_mode_manager();

CASE process_get_mode(prc) OF
	MODE_ABSENT:
		IF axis_get_mode(axis) = MODE_TEST
		THEN
			safety_integrated_series_close(csp_transfer_main_safety_drives_SD41100.chA_smes_sis);
		END_IF
		RETURN;
	MODE_INACTIVE:
		RETURN;
	MODE_TEST:
		_handle_process_test();
END_CASE

(********************************* BODY *********************************)
axis.actual_torque := (axis.actual_current * Torque_force_constant)/1000;

(* Sets torque Limit *)
IF torque_limit <> torque_limit_old
THEN
	IF soe_drive_channel_write_parameter(
		channel:= csp_transfer_accumulator_lift.axis.soe_drive_channel, 
		idn:= S_0_IDN + 92, 
		data_element:= soe_drive_element_value, 
		data_source:= ADR(torque_limit), 
		data_lenght:= SIZEOF(torque_limit),
		CONVERSION_this:= csp_transfer_accumulator_lift.axis.soe_drive^) = SOE_DRIVE_RETURN_VALUE_DONE
	THEN
		torque_limit_old := torque_limit;
	END_IF
END_IF

(* Connection Done Test *)
IF connection_done
THEN 
	motorization_conditioner_start_done(connection_done_motcond);
END_IF

(* CLEARS CONNECTION AND PHASE ERRORS *)
IF 	machine_is_stopped(csp.mch)
	OR machine_is_stop_emergency_active(csp.mch)
	OR machine_is_ready(csp.mch)
	OR csp_main_services_pushbuttons.i_reset_button
THEN
	connection_error := FALSE;
	phase_error := FALSE;
END_IF

(* RESETS AXES IF PHASE DONE AND CONNECTION DONE AND DISABLED *)
IF 	phase_done
	AND connection_done
	AND axis_is_disabled(axis)
THEN
	phase_done := FALSE;
	connection_done := FALSE;
END_IF


(* CAM CHANGE/CHECK LOGIC *)
IF 	phase_edge(csp_transfer_crosspusher_virtualMaster.cam_change_check_ph) (* CROSSPUSHER VIRTUAL AT CHECK PHASE DEG *)
	AND connection_status = CSP_TRANSFER_CROSSPUSHER_STATUS_CONNECTION_CHECK_CHANGE_CAM
THEN	
	IF run_test 
	OR
	(
	csp_transfer_upstacker.stack_made (* UPSTACKER MADE CORRECT AMOUNT OF STACK *)
	AND csp_transfer_crosspusher_horizontal.at_upstack (* VERIFIES THE HORIZONTAL IS AT THE UPSTACKER BEFORE RUNNING *)
	AND NOT csp_transfer_upstacker.stack_at_loader (* MAKES SURE A STACK IS NOT ALREADY AT THE LOADER *)
	)
	THEN 
		run := TRUE;
	ELSE
		dwell := TRUE;
	END_IF
END_IF

(* DWELL CAM BECAUSE LOADER NOT CLEAR - IMMEDIATELY *)
IF active_cam = TRANSFER_ACCUMULATOR_LIFT_RUN
	AND csp_transfer_crosspusher.loader_status = csp_transfer_crosspusher_loader_clear_status.NOT_CLEAR 
THEN
	connection_status_next := CSP_TRANSFER_CROSSPUSHER_STATUS_CONNECTION_IMMEDIATE_CHANGE;
	connection_status := CSP_TRANSFER_CROSSPUSHER_STATUS_CONNECTION_IMMEDIATE_CHANGE;
END_IF

(* ERROR HANDLING FOR CAM ERROR *)
IF active_cam = 0
THEN 
	active_cam := DWELL_CAM;
END_IF

(* TELLS THE FOLLOWER WHAT THE PROFILE SHOULD BE ON A CLEARED LOAD *)
IF csp_transfer_upstacker.stack_removed_from_upstack
THEN
	active_cam := DWELL_CAM;
END_IF

(* MAIN ACTIONS IN POU *)
phase();
connection();
_set_runtime_properties();

(************************************************************************)

_handle_messages();

_write_output();

ACTION _handle_messages:
;
END_ACTION

ACTION _handle_process_test:
;
END_ACTION

ACTION _mode_manager:
IF process_mode_req_is_pending(prc)
THEN
    process_apply_mode_req_first_step(prc);
    CASE process_get_mode(prc) OF
        MODE_TO_ABSENT:
			;
        MODE_TO_INACTIVE:
			;
        MODE_TO_TEST:
			;
        MODE_TO_OPERATIONAL:
			;
    END_CASE
    process_apply_mode_req_second_step(prc);
END_IF
END_ACTION

ACTION _object_manager:
IF objects_initialization()
THEN
	sub_process_init(
		object_name					:= 'csp_transfer_accumulator_lift.prc', 
		process						:= csp_transfer_accumulator.prc, 
		CONVERSION_this				:= prc);
		
	prc_path 						:= process_get_path(prc);
	
	axis_init(
		object_name					:= CONCAT(prc_path, '_axis'), 
		axis_type					:= AXIS_TYPE_SERVO, 
		encoder_scaling_factor		:= G_SERVO_ENCODER_SCALING_FACTOR_DEGPINC,
		modulo						:= G_MODULO_360_DEG, 
		process						:= prc, 
		CONVERSION_this				:= axis);
		
	axis_init_absolute_encoder_preset(	
		position					:=	0,
		CONVERSION_this				:=	axis);
	
	axis_set_max_dynamic(
		reference_velocity			:=	MOTOR_MAX_VELOCITY_DEGPS,
		velocity					:=	MOTOR_MAX_VELOCITY_DEGPS,
		acceleration				:=	MOTOR_MAX_ACCELLERATION_DEGPS2,
		deceleration				:=	MOTOR_MAX_DECELLERATION_DEGPS2,
		jerk						:=	MOTOR_MAX_JERK_DEGPS3,
		following_error				:=	MOTOR_MAX_FOLLOWING_ERROR_DEG,
		CONVERSION_this				:=	axis);
	
	axis_add_soe_drive(
		channel						:=	SOE_DRIVE_CHANNEL_A,
		soe_drive					:=	csp_transfer_main_drives.SD41100_drv,
		CONVERSION_this				:=	axis);
		
	process_message_init(
		object_name					:=	CONCAT(prc_path, '_phase_faulted_aem'), 
		behaviour					:=	MESSAGE_BEHAVIOUR_EVENT,
		reset_timeout				:=	0,
		disableable					:=	TRUE,
		individual_reset			:=	FALSE,
		machine_reaction			:=	MACHINE_REACTION_NORMAL_STOP,
		typology					:=	MESSAGE_TYPOLOGY_ABNORMAL,
		process						:=	prc,
		CONVERSION_this				:=	phase_faulted_aem);
	
	timer_init(
		object_name					:= CONCAT(prc_path, 'phase_time_out_tmr'),
		process						:= prc,
		CONVERSION_this				:= phase_time_out_tmr);
		
	process_message_init(
		object_name					:=	CONCAT(prc_path, 'debug_immediate_stop_aem'), 
		behaviour					:=	MESSAGE_BEHAVIOUR_STATE,
		reset_timeout				:=	0,
		disableable					:=	TRUE,
		individual_reset			:=	FALSE,
		machine_reaction			:=	MACHINE_REACTION_NORMAL_STOP,
		typology					:=	MESSAGE_TYPOLOGY_ABNORMAL,
		process						:=	prc,
		CONVERSION_this				:=	debug_immediate_stop_aem);
		
	timer_init(
		object_name					:= CONCAT(prc_path, 'connection_time_out_tmr'),
		process						:= prc,
		CONVERSION_this				:= connection_time_out_tmr);
		
		
	process_message_init(
		object_name					:=	CONCAT(prc_path, '_connection_faulted_aem'), 
		behaviour					:=	MESSAGE_BEHAVIOUR_EVENT,
		reset_timeout				:=	0,
		disableable					:=	TRUE,
		individual_reset			:=	FALSE,
		machine_reaction			:=	MACHINE_REACTION_NORMAL_STOP,
		typology					:=	MESSAGE_TYPOLOGY_ABNORMAL,
		process						:=	prc,
		CONVERSION_this				:=	connection_faulted_aem);
		
	motorization_conditioner_init(
		object_name					:=	CONCAT(prc_path, 'connection_done_motcond'),
		velocity_limit				:=	0.0,
		velocity_limit_active		:=	FALSE,
		idle_handshake_active		:=	FALSE,
		execute_handshake_active	:=	TRUE,
		hold_handshake_active		:=	FALSE,
		suspend_handshake_active	:=	FALSE,
		complete_handshake_active	:=	FALSE,
		abort_handshake_active		:=	FALSE,
		stop_handshake_active		:=	FALSE,
		origin						:=	MOTORIZATION_CONDITIONER_ORIGIN_INTERNAL,
		manager						:=	csp_main_motorization_manager.motm,
		process						:=	prc,
		CONVERSION_this				:=	connection_done_motcond);	

	jog_manager_add_axis(
		list_index					:= SMTR41103_TRANSFER_ACCUMULATOR_LIFT,
		axis						:= axis,
		master_axis					:= FALSE,
		jog_type					:= JOG_TYPE_ROTATIVE,
		sw_limit_positive			:= 0,
		sw_limit_negative			:= 0,
		CONVERSION_this				:= csp_main_jogManager.jog_manager_real);		
		
		
	IF csp_main_configurator.Physical_hw
	THEN
		axis_add_safety_integrated_series(
			safety_integrated_series 	:= csp_transfer_main_safety_drives_SD41100.chA_smes_sis,
			CONVERSION_this				:= axis);
	END_IF

END_IF

IF objects_running()
THEN
	process_cycle(prc);
	
	axis_cycle(axis);
	
	motorization_conditioner_cycle(connection_done_motcond);
END_IF
END_ACTION

ACTION _read_process_image:
;
END_ACTION

ACTION _read_var_input:
;
END_ACTION

ACTION _set_runtime_properties:
(* Cam management *)
IF 	connection_done
THEN
	active_cam := axis.engaged_cam.cam_id;
END_IF

enable_delay(IN:=axis_is_ready_to_enable(axis) , PT:=T#2S , Q=> servo_on_condition , ET=> );
END_ACTION

ACTION _write_output:
;
END_ACTION

ACTION connection:
connection_conditions :=	
	axis_is_ok(FALSE, axis)
	AND
	servo_on_condition
	AND
	NOT process_message_is_on(connection_faulted_aem)
	AND
	phase_done;

(* connection_done reset *)
IF	connection_done
	AND	
	NOT connection_conditions
	AND
	NOT csp.o_machine_is_running
THEN
	connection_done := FALSE;
END_IF

(* Exit conditions *)
IF	NOT connection_conditions 
	AND
	NOT motorization_manager_is_stopping(csp_main_motorization_manager.motm)	
THEN	
	connection_status_next := CSP_TRANSFER_CROSSPUSHER_STATUS_CONNECTION_ERROR;
	connection_status := connection_status_next;	
END_IF

(*************** MACHINE STATUS ***************)
CASE connection_status OF

	CSP_TRANSFER_CROSSPUSHER_STATUS_CONNECTION_START:	(* Start connection *)
	
		IF	motorization_manager_is_starting(csp_main_motorization_manager.motm) //TODOPZ: da decidere a che livello usare le variabili di i e o: wn_feeding.i_motorization_is_starting?					
		THEN
			connection_running := TRUE;
			connection_status_next := CSP_TRANSFER_CROSSPUSHER_STATUS_CONNECTION_ENGAGE;
		END_IF
		
		
	CSP_TRANSFER_CROSSPUSHER_STATUS_CONNECTION_ENGAGE:		
		
		IF active_cam = TRANSFER_ACCUMULATOR_LIFT_RUN
		THEN
			master_offset_phase := csp_transfer_crosspusher_virtualMaster.axis.actual_modulo_position; 
			master_engage_mode := AXIS_CAM_ENGAGE_RELATIVE;
		ELSE
			master_offset_phase := 0.0;
			master_engage_mode := AXIS_CAM_ENGAGE_ABSOLUTE;
		END_IF
	
		axis_engage_cam(
			cam_id							:=	active_cam,	
			master_engage_mode				:=	master_engage_mode,
			slave_engage_mode				:=	AXIS_CAM_ENGAGE_ABSOLUTE,
			activation_mode					:=	AXIS_CAM_ACTIVATION_IMMEDIATELY,
			activation_position				:=	0.0,
			master_scaling_mode				:=	AXIS_CAM_SCALING_MODE_USER_DEFINED,
			slave_scaling_mode				:=	AXIS_CAM_SCALING_MODE_USER_DEFINED,
			master_offset					:=	master_offset + master_offset_phase,
			slave_offset					:=	slave_offset,
			master_scaling					:=	master_scaling,
			slave_scaling					:=	slave_scaling,
			interpolation_type				:=	AXIS_CAM_INTERPOLATION_SPLINE,	 
			master							:=	csp_transfer_crosspusher_virtualMaster.axis,
			CONVERSION_this					:=	axis);
		
		connection_status_next:= CSP_TRANSFER_CROSSPUSHER_STATUS_CONNECTION_ENGAGED;
	
		
	CSP_TRANSFER_CROSSPUSHER_STATUS_CONNECTION_ENGAGED:
	
		IF 	axis_is_cam_engaged(axis) 
		THEN				
			IF	active_cam <> next_cam
			THEN							
				connection_status_next := CSP_TRANSFER_CROSSPUSHER_STATUS_CONNECTION_CHANGE_CAM;
			ELSE
				connection_status_next:= CSP_TRANSFER_CROSSPUSHER_STATUS_CONNECTION_DONE;
			END_IF
		END_IF
		
		
	CSP_TRANSFER_CROSSPUSHER_STATUS_CONNECTION_CHECK_CHANGE_CAM:						
		
		IF dwell
			THEN			
				CASE active_cam OF
					
					DWELL_CAM:
						dwell := FALSE;
	
					TRANSFER_ACCUMULATOR_LIFT_RUN:
					
						next_cam := DWELL_CAM;	
						dwell := FALSE; 					
						
				END_CASE				
		END_IF
		
		IF run
			AND (
				(* USED FOR 2 STACK TO QUEUE MOVE TO LOAD *)
				(csp_main_brand.case_pattern.case_pattern_W = 2
				AND csp_transfer_virtualMaster.section_0_180) (* PHASE CHECK BASED OFF OF STACK COUNT *)
			OR 
				(* USED FOR 3 STACK TO QUEUE MOVE TO LOAD *)
				(csp_main_brand.case_pattern.case_pattern_W = 3
				AND csp_transfer_virtualMaster.section_120_240)
			)
		THEN
		
			CASE active_cam OF
				
				DWELL_CAM:
					next_cam := TRANSFER_ACCUMULATOR_LIFT_RUN;
					run := FALSE;

				TRANSFER_ACCUMULATOR_LIFT_RUN:
					run := FALSE;
					
			END_CASE
		END_IF
					
		IF	(active_cam <> next_cam)
			AND 
			connection_conditions
		THEN							
			connection_status_next := CSP_TRANSFER_CROSSPUSHER_STATUS_CONNECTION_CHANGE_CAM;
		END_IF
			
		IF	NOT connection_motorization_moving
		THEN
			connection_status_next := CSP_TRANSFER_CROSSPUSHER_STATUS_CONNECTION_DONE;
		END_IF
	
		
	CSP_TRANSFER_CROSSPUSHER_STATUS_CONNECTION_CHANGE_CAM:	
		
		axis_engage_cam(
				cam_id							:=	next_cam,	
				master_engage_mode				:=	AXIS_CAM_ENGAGE_RELATIVE,
				slave_engage_mode				:=	AXIS_CAM_ENGAGE_RELATIVE,
				activation_mode					:=	AXIS_CAM_ACTIVATION_NEXT_CYCLE,
				activation_position				:=	0,
				master_scaling_mode				:=	AXIS_CAM_SCALING_MODE_USER_DEFINED,
				slave_scaling_mode				:=	AXIS_CAM_SCALING_MODE_USER_DEFINED,
				master_offset					:=	master_offset, 
				slave_offset					:=	slave_offset,
				master_scaling					:=	master_scaling,
				slave_scaling					:=	slave_scaling,
				interpolation_type				:=	AXIS_CAM_INTERPOLATION_SPLINE,	 
				master							:=	csp_transfer_crosspusher_virtualMaster.axis,
				CONVERSION_this					:=	axis);	
	
		IF	motorization_manager_is_starting(csp_main_motorization_manager.motm)
		THEN
			connection_status_next := CSP_TRANSFER_CROSSPUSHER_STATUS_CONNECTION_DONE;
		ELSE
			IF axis_is_cam_engaged(axis)
			THEN
				connection_status_next := CSP_TRANSFER_CROSSPUSHER_STATUS_CONNECTION_WAIT_NEW_CAM;
			END_IF
		END_IF
		
		
	CSP_TRANSFER_CROSSPUSHER_STATUS_CONNECTION_IMMEDIATE_CHANGE:
	
		axis_engage_cam(
			cam_id							:=	DWELL_CAM,	
			master_engage_mode				:=	AXIS_CAM_ENGAGE_ABSOLUTE,
			slave_engage_mode				:=	AXIS_CAM_ENGAGE_RELATIVE,
			activation_mode					:=	AXIS_CAM_ACTIVATION_IMMEDIATELY,
			activation_position				:=	0,
			master_scaling_mode				:=	AXIS_CAM_SCALING_MODE_USER_DEFINED,
			slave_scaling_mode				:=	AXIS_CAM_SCALING_MODE_USER_DEFINED,
			master_offset					:=	csp_transfer_crosspusher_virtualMaster.axis.actual_position, 
			slave_offset					:=	slave_offset,
			master_scaling					:=	master_scaling,
			slave_scaling					:=	slave_scaling,
			interpolation_type				:=	AXIS_CAM_INTERPOLATION_SPLINE,	 
			master							:=	csp_transfer_crosspusher_virtualMaster.axis,
			CONVERSION_this					:=	axis);	
			
		next_cam := DWELL_CAM;
		active_cam := DWELL_CAM;
					
		IF	motorization_manager_is_starting(csp_main_motorization_manager.motm)
		THEN
			connection_status_next := CSP_TRANSFER_CROSSPUSHER_STATUS_CONNECTION_DONE;
		ELSE
			IF csp_transfer_crosspusher.loader_clear
			THEN
				connection_status_next := CSP_TRANSFER_CROSSPUSHER_STATUS_CONNECTION_WAIT_NEW_CAM;
			END_IF
		END_IF	
				
	
	CSP_TRANSFER_CROSSPUSHER_STATUS_CONNECTION_WAIT_NEW_CAM:
	
		IF	active_cam = next_cam
		THEN
			CASE next_cam OF
				DWELL_CAM:
					activation_position := next_activation_position;
				
				FORWARD_CAM:
					activation_position := 0;
					
			END_CASE
			connection_status_next := CSP_TRANSFER_CROSSPUSHER_STATUS_CONNECTION_CHECK_CHANGE_CAM;
		END_IF
		
		IF	NOT connection_motorization_moving
		THEN
			connection_status_next := CSP_TRANSFER_CROSSPUSHER_STATUS_CONNECTION_DONE;
		END_IF
		
		
	CSP_TRANSFER_CROSSPUSHER_STATUS_CONNECTION_DONE:    (* Connection done *)  
     
        connection_running := FALSE;
        connection_done := TRUE;
       
        motorization_conditioner_start_done(connection_done_motcond);
		IF	csp.o_machine_is_running
		THEN                       
			IF    active_cam <> next_cam
			THEN
				connection_status_next := CSP_TRANSFER_CROSSPUSHER_STATUS_CONNECTION_WAIT_NEW_CAM;
			ELSE
				connection_status_next := CSP_TRANSFER_CROSSPUSHER_STATUS_CONNECTION_CHECK_CHANGE_CAM;
			END_IF
        END_IF
       
       	
	CSP_TRANSFER_CROSSPUSHER_STATUS_CONNECTION_ERROR:	(* Connection error *)
	
		IF 	connection_running
			OR NOT axis_is_ok(FALSE, axis)
		THEN
			axis_disable(axis);	
			connection_error := TRUE;					
		END_IF
		connection_running	:= FALSE;
		connection_done 	:= FALSE;	
		
		IF	connection_conditions
		THEN		
			connection_status_next := CSP_TRANSFER_CROSSPUSHER_STATUS_CONNECTION_START;
		END_IF
		
END_CASE

IF 	NOT debug_state_machine
	OR
	debug_connection_machine_one_step	
THEN
	connection_status := connection_status_next;
	debug_connection_machine_one_step := FALSE;
END_IF

connection_motorization_moving	:= 
	motorization_manager_is_starting(csp_main_motorization_manager.motm)
	OR
	motorization_manager_is_execute(csp_main_motorization_manager.motm)
	OR
	motorization_manager_is_stopping(csp_main_motorization_manager.motm)
	OR
	motorization_manager_is_suspended(csp_main_motorization_manager.motm)
	OR
	motorization_manager_is_suspending(csp_main_motorization_manager.motm)
	OR
	motorization_manager_is_unsuspending(csp_main_motorization_manager.motm)
	OR 
	motorization_manager_is_holding(csp_main_motorization_manager.motm)
	OR
	motorization_manager_is_held(csp_main_motorization_manager.motm)
	OR
	motorization_manager_is_unholding(csp_main_motorization_manager.motm);
	
(* Connection timeout *)
IF	(connection_running
	AND NOT debug_state_machine)	
	OR connection_error
THEN
	IF	timer_is_expired(connection_time_out_tmr)
	THEN
		process_message_set(1, connection_status, 0, connection_faulted_aem);
	END_IF
ELSE
	timer_restart(10000, connection_time_out_tmr);
END_IF
END_ACTION

ACTION phase:
phase_conditions :=
	axis_is_ok(FALSE, axis)
	AND
	process_is_ready(prc)
	AND
	process_subtree_is_ready(prc)
	AND
	servo_on_condition
	AND				
	NOT csp_transfer_main_brand.cam_data_changed
	AND
	NOT disable_req
	AND						
	NOT jog_manager_is_jog_axis_active(SMTR41103_TRANSFER_ACCUMULATOR_LIFT, csp_main_jogManager.jog_manager_real);				
	
(* phase_done reset *)
IF	phase_done
	AND
	NOT phase_conditions
	AND 
	NOT csp.o_machine_is_running
THEN
	axis_disable(axis);
	
	phase_done:= FALSE;
END_IF

(* Exit condition *)
IF 	NOT phase_conditions
THEN
	phase_status_next := CSP_TRANSFER_CROSSPUSHER_PHASE_STATUS_ERROR;
	phase_status := phase_status_next;	
END_IF

(*************** MACHINE STATUS ***************)
CASE phase_status OF

	CSP_TRANSFER_CROSSPUSHER_PHASE_STATUS_START:	(* Start phasing *)
	
		IF	motorization_manager_is_starting(csp_main_motorization_manager.motm) 					
			AND csp_transfer_crosspusher_virtualMaster.phase_done
			AND csp_transfer_crosspusher_virtualMaster.connection_done
		THEN
			phase_running := TRUE;			
			phase_status_next := CSP_TRANSFER_CROSSPUSHER_PHASE_STATUS_DISABLE;
		END_IF
		
				
	CSP_TRANSFER_CROSSPUSHER_PHASE_STATUS_DISABLE:
	
		axis_disable(axis);				
		IF 	axis_is_disabled(axis)
		THEN
			phase_status_next := CSP_TRANSFER_CROSSPUSHER_PHASE_STATUS_ENABLE;
		END_IF
		
		
	CSP_TRANSFER_CROSSPUSHER_PHASE_STATUS_ENABLE:
	
		axis_enable(axis);		
		IF 	axis_is_enabled(axis)
		THEN
			phase_status_next := CSP_TRANSFER_CROSSPUSHER_PHASE_STATUS_ENABLED;
		END_IF
		
		
	CSP_TRANSFER_CROSSPUSHER_PHASE_STATUS_ENABLED:
	
		IF 	axis_is_standstill(axis) 
		THEN
			phase_status_next := CSP_TRANSFER_CROSSPUSHER_PHASE_STATUS_CALCULATE_SLAVE_POSITION_REQUEST;								
		END_IF
		
		
	CSP_TRANSFER_CROSSPUSHER_PHASE_STATUS_CALCULATE_SLAVE_POSITION_REQUEST:
	
		slave_position_has_been_calculated := FALSE;
	
		(* Gets the position of the master axis *)
		axis_calculate_cam_slave_master_position_deg := 
			LMOD(axis_get_actual_modulo_position(csp_transfer_crosspusher_virtualMaster.axis)
			+ home_position_master_offset_deg, G_MODULO_360_DEG);
			
		(* Gets cam data for slave axis to master *)
		IF axis_calculate_cam_slave_dynamics_data(
			cam_id := active_cam,
			master_scaling := master_scaling,
			master_position := axis_calculate_cam_slave_master_position_deg,
			slave_scaling := slave_scaling,
			CONVERSION_this := axis)
		THEN
			phase_status_next := CSP_TRANSFER_CROSSPUSHER_PHASE_STATUS_CALCULATING_SLAVE_POSITION;
		END_IF
	
		
	CSP_TRANSFER_CROSSPUSHER_PHASE_STATUS_CALCULATING_SLAVE_POSITION:
	
		IF axis_cam_slave_dynamics_data_calculated(axis)
		THEN
			axis_calculated_cam_slave_position_deg := axis_get_cam_slave_dynamics_position(axis);
			slave_position_has_been_calculated := TRUE;
			phase_status_next := CSP_TRANSFER_PHASE_STATUS_REQUEST;				
		END_IF
		
		
	CSP_TRANSFER_PHASE_STATUS_REQUEST:
		
		IF	axis_is_standstill(axis)
		THEN
			 axis_move_absolute(
				position 		:= axis_calculated_cam_slave_position_deg,
				velocity 		:= phase_velocity_degps,
				direction		:= AXIS_SHORTEST_WAY,
				acceleration 	:= MOTOR_MAX_ACCELLERATION_DEGPS2,
				deceleration 	:= MOTOR_MAX_DECELLERATION_DEGPS2, 
				jerk 			:= MOTOR_MAX_JERK_DEGPS3, 
				buffer_mode 	:= AXIS_BUFFER_MODE_BUFFERED,
				CONVERSION_this := axis
				); 			
		END_IF

		IF axis_is_absolute_moving(axis)
		THEN
			phase_status_next	:=	CSP_TRANSFER_PHASE_STATUS_PHASING;
		END_IF

		
	CSP_TRANSFER_PHASE_STATUS_PHASING:

		IF axis_is_standstill(axis)
		THEN
			phase_status_next	:=	CSP_TRANSFER_CROSSPUSHER_STATUS_PHASED;
		END_IF

		
	CSP_TRANSFER_CROSSPUSHER_STATUS_PHASED:

		IF engage_enable
		THEN
			phase_status_next := CSP_TRANSFER_CROSSPUSHER_PHASE_STATUS_DONE;
		END_IF
		
		
	CSP_TRANSFER_CROSSPUSHER_PHASE_STATUS_DONE:	(* Phase done *)
			
		phase_running := FALSE;
		phase_done := TRUE;				
	
		
	CSP_TRANSFER_CROSSPUSHER_PHASE_STATUS_ERROR:	(* Phase error *)
	
		IF	phase_running
		THEN
			phase_error := TRUE;
			axis_disable(axis);									
		END_IF
		phase_running := FALSE;
		
		IF	phase_conditions 	
		THEN
			phase_status_next := CSP_TRANSFER_CROSSPUSHER_PHASE_STATUS_START;
		END_IF
		
END_CASE

IF 	NOT debug_state_machine
	OR
	debug_phase_machine_one_step	
THEN
	phase_status := phase_status_next;
	debug_phase_machine_one_step := FALSE;
END_IF

(* Phasing timeout *)
IF (phase_running
AND NOT debug_state_machine)
OR phase_error
THEN
	IF	timer_is_expired(phase_time_out_tmr)
	THEN
		process_message_set(1, phase_status, 0, phase_faulted_aem);
	END_IF
ELSE
	timer_restart(30000, phase_time_out_tmr);
END_IF
END_ACTION

END_PROGRAM

// ---- Application/CSP/Main/_Tasks/_csp_main_highest.TcPOU
(*********************************** G.D S.p.A. - Technical Department ***********************************
============= PROGRAM INFO ============
FOLDER:             TBD
MACHINES INVOLVED:  TBD 

============= DESCRIPTION =============
csp main interface program

============= REVISIONS ===============
Date		Version	 	Author      	Description             
----------	-------		------------  	--------------------------------------------
2019/09/27 	0000.00	 	M.Grasso		Creation of the PRG

**********************************************************************************************************)
PROGRAM _csp_main_highest
VAR
END_VAR

(*MAIN*)
 IF	objects_running()  (*//Nick*)
THEN
	quality_checks_cycle();
END_IF;

	(*Drives*)
	csp_main_drives();
	(*Motorization*)
	csp_main_motorization_manager();
	//csp_main_motorization();	
	csp_main_motorization_virtualManager();

	(*Services*)
	
	(*Interface*)
	csp_main_interface();
	csp_main_interface_upstream();
	csp_main_interface_downstream();
	(*Safety*)

END_PROGRAM

// ---- Application/CSP/Main/Drives/csp_main_drives.TcPOU
(*********************************** G.D S.p.A. - Technical Department ***********************************
============= PROGRAM INFO ============
FOLDER:             TBD
MACHINES INVOLVED:  TBD 

============= DESCRIPTION =============

============= REVISIONS ===============
Date		Version	 	Author      	Description             
----------	-------		------------  	--------------------------------------------
2019/04/24 	0000.00	 	M.Grasso			Creation of the PRG

**********************************************************************************************************)
(*$R
	process_ref := prc;
$*)
PROGRAM csp_main_drives
VAR
	prc:						process;
	prc_path:					STRING;
	
		
END_VAR

VAR CONSTANT
	INCOHERENCE_TIMEOUT_MS:		INT := 2000;
END_VAR

_read_var_input();

_object_manager();

IF NOT objects_running()
THEN
	RETURN;	
END_IF

_read_process_image();

_mode_manager();

CASE process_get_mode(prc) of
	MODE_ABSENT,
	MODE_INACTIVE:
		RETURN;
	MODE_TEST:
		_handle_process_test();
END_CASE

_set_runtime_properties();

(********************************* BODY *********************************)

(************************************************************************)

_handle_messages();

_write_output();

ACTION _handle_messages:
;
END_ACTION

ACTION _handle_process_test:
;
END_ACTION

ACTION _mode_manager:
IF process_mode_req_is_pending(prc)
THEN
    process_apply_mode_req_first_step(prc);
    CASE process_get_mode(prc) OF
        MODE_TO_ABSENT:
			;
        MODE_TO_INACTIVE:
			;
        MODE_TO_TEST:
			;
        MODE_TO_OPERATIONAL:
			;
    END_CASE
    process_apply_mode_req_second_step(prc);
END_IF
END_ACTION

ACTION _object_manager:
IF objects_initialization()
THEN
	sub_process_init(
		object_name					:= 'csp_main_drives.prc', 
		process						:= csp_main.prc, 
		CONVERSION_this				:= prc);
		
	prc_path 						:= process_get_path(prc);

END_IF

IF objects_running()
THEN
	process_cycle(prc);
	
	
END_IF
END_ACTION

ACTION _read_process_image:
;
END_ACTION

ACTION _read_var_input:
;
END_ACTION

ACTION _set_runtime_properties:
;
END_ACTION

ACTION _write_output:
;
END_ACTION

END_PROGRAM

// ---- Application/CSP/Main/Interface/Upstream/csp_main_interface_upstream.TcPOU
(*********************************** G.D S.p.A. - Technical Department ***********************************
============= PROGRAM INFO ============
FOLDER:             TBD
MACHINES INVOLVED:  TBD 

============= DESCRIPTION =============
csp - Upstream interface

============= REVISIONS ===============
Date		Version	 	Author      	Description             
----------	-------		------------  	--------------------------------------------
2019/10/07 	0000.00	 	W. Gerstner		Creation of the PRG

**********************************************************************************************************)
(*$R
	process_ref := prc;
$*)
PROGRAM csp_main_interface_upstream
VAR
	prc:					process;
	prc_path:				STRING;	

END_VAR

_read_var_input();

_object_manager();

IF NOT objects_running()
THEN
	RETURN;	
END_IF

_read_process_image();

_mode_manager();

CASE process_get_mode(prc) of
	MODE_ABSENT,
	MODE_INACTIVE:
		RETURN;
	MODE_TEST:
		_handle_process_test();
END_CASE

_set_runtime_properties();

(********************************* BODY *********************************)

(************************************************************************)

_handle_messages();

_write_output();

ACTION _handle_messages:
;
END_ACTION

ACTION _handle_process_test:
;
END_ACTION

ACTION _mode_manager:
IF process_mode_req_is_pending(prc)
THEN
    process_apply_mode_req_first_step(prc);
    CASE process_get_mode(prc) OF
        MODE_TO_ABSENT:
			;
        MODE_TO_INACTIVE:
			;
        MODE_TO_TEST:
			;
        MODE_TO_OPERATIONAL:
			;
    END_CASE
    process_apply_mode_req_second_step(prc);
END_IF
END_ACTION

ACTION _object_manager:
IF objects_initialization()
THEN
	sub_process_init(
		object_name					:= 'csp_main_interface_upstream.prc', 
		process						:= csp_main_interface.prc, 
		CONVERSION_this				:= prc);
		
	prc_path 						:= process_get_path(prc);
END_IF

IF objects_running()
THEN
	process_cycle(prc);
END_IF
END_ACTION

ACTION _read_process_image:
;
END_ACTION

ACTION _read_var_input:
;
END_ACTION

ACTION _set_runtime_properties:
;
END_ACTION

ACTION _write_output:
;
END_ACTION

END_PROGRAM

// ---- Application/CSP/Main/Interface/Downstream/csp_main_interface_downstream.TcPOU
(*********************************** G.D S.p.A. - Technical Department ***********************************
============= PROGRAM INFO ============
FOLDER:             TBD
MACHINES INVOLVED:  TBD 

============= DESCRIPTION =============
csp - Downstream Interface

============= REVISIONS ===============
Date		Version	 	Author      	Description             
----------	-------		------------  	--------------------------------------------
2019/10/07 	0000.00	 	W. Gerstner		Creation of the PRG

**********************************************************************************************************)
(*$R
	process_ref := prc;
$*)
PROGRAM csp_main_interface_downstream
VAR
	prc:					process;
	prc_path:				STRING;	

END_VAR

_read_var_input();

_object_manager();

IF NOT objects_running()
THEN
	RETURN;	
END_IF

_read_process_image();

_mode_manager();

CASE process_get_mode(prc) of
	MODE_ABSENT,
	MODE_INACTIVE:
		RETURN;
	MODE_TEST:
		_handle_process_test();
END_CASE

_set_runtime_properties();

(********************************* BODY *********************************)

(************************************************************************)

_handle_messages();

_write_output();

ACTION _handle_messages:
;
END_ACTION

ACTION _handle_process_test:
;
END_ACTION

ACTION _mode_manager:
IF process_mode_req_is_pending(prc)
THEN
    process_apply_mode_req_first_step(prc);
    CASE process_get_mode(prc) OF
        MODE_TO_ABSENT:
			;
        MODE_TO_INACTIVE:
			;
        MODE_TO_TEST:
			;
        MODE_TO_OPERATIONAL:
			;
    END_CASE
    process_apply_mode_req_second_step(prc);
END_IF
END_ACTION

ACTION _object_manager:
IF objects_initialization()
THEN
	sub_process_init(
		object_name						:= 'csp_main_interface_downstream.prc', 
		process							:= csp_main_interface.prc, 
		CONVERSION_this					:= prc);
		
	prc_path 							:= process_get_path(prc);
END_IF

IF objects_running()
THEN
	process_cycle(prc);
END_IF
END_ACTION

ACTION _read_process_image:
;
END_ACTION

ACTION _read_var_input:
;
END_ACTION

ACTION _set_runtime_properties:
;
END_ACTION

ACTION _write_output:
;
END_ACTION

END_PROGRAM

// ---- Application/CSP/Customer Interface/_Tasks/_csp_customerInterfaces_highest.TcPOU
(*********************************** G.D S.p.A. - Technical Department ***********************************
============= PROGRAM INFO ============
FOLDER:             TBD
MACHINES INVOLVED:  TBD 

============= DESCRIPTION =============
Low task

============= REVISIONS ===============
Date		Version	 	Author      	Description             
----------	-------		------------  	--------------------------------------------
2019/03/28 	0000.00	 	CEC 			Creation of the PRG

**********************************************************************************************************)

PROGRAM _csp_customerInterfaces_highest
VAR
END_VAR

;

END_PROGRAM

// ---- Application/_Tasks/_lowest.TcPOU
(*********************************** G.D S.p.A. - Technical Department ***********************************
============= PROGRAM INFO ============
FOLDER:             TBD
MACHINES INVOLVED:  TBD 

============= DESCRIPTION =============
Highest task

============= REVISIONS ===============
Date		Version	 	Author      	Description             
----------	-------		------------  	--------------------------------------------
2019/04/05 	0000.00	 	G.Cera 			Creation of the PRG

**********************************************************************************************************)
{attribute 'TcCallAfterOutputUpdate'}
PROGRAM _lowest
VAR
END_VAR

(* APPLICATION *)
framework_lowesttask_begin();


_csp_lowest();

//dbg_lowest();

framework_lowesttask_end();

END_PROGRAM

// ---- Application/CSP/_Tasks/_csp_lowest.TcPOU
(*********************************** G.D S.p.A. - Technical Department ***********************************
============= PROGRAM INFO ============
FOLDER:             TBD
MACHINES INVOLVED:  TBD 

============= DESCRIPTION =============
CSP: lowest task

============= REVISIONS ===============
Date		Version	 	Author      	Description             
----------	-------		------------  	--------------------------------------------
2019/04/05 	0000.00	 	G.Cera 			Creation of the PRG

**********************************************************************************************************)

PROGRAM _csp_lowest
VAR
END_VAR

_csp_case_lowest();

_csp_transfer_lowest();

_csp_main_lowest();

_csp_customerInterfaces_lowest();

END_PROGRAM

// ---- Application/CSP/Case/_Tasks/_csp_case_lowest.TcPOU
(*********************************** G.D S.p.A. - Technical Department ***********************************
============= PROGRAM INFO ============
FOLDER:             TBD
MACHINES INVOLVED:  TBD 

============= DESCRIPTION =============
csp main interface program

============= REVISIONS ===============
Date		Version	 	Author      	Description             
----------	-------		------------  	--------------------------------------------
2019/09/27 	0000.00	 	M.Grasso		Creation of the PRG

**********************************************************************************************************)
PROGRAM _csp_case_lowest
VAR
END_VAR

_csp_case_closing_lowest();

_csp_case_discharge_lowest();

_csp_case_feed_lowest();

_csp_case_flapControl_lowest();

_csp_case_glue_lowest();

_csp_case_loader_lowest();

_csp_case_openFlap_lowest();

_csp_case_main_lowest();

_csp_case_topRail_lowest();

_csp_case_transport_lowest();

END_PROGRAM

// ---- Application/CSP/Case/Closing/_Tasks/_csp_case_closing_lowest.TcPOU
(*********************************** G.D S.p.A. - Technical Department ***********************************
============= PROGRAM INFO ============
FOLDER:             TBD
MACHINES INVOLVED:  TBD 

============= DESCRIPTION =============
csp main interface program

============= REVISIONS ===============
Date		Version	 	Author      	Description             
----------	-------		------------  	--------------------------------------------
2019/09/27 	0000.00	 	M.Grasso		Creation of the PRG

**********************************************************************************************************)
PROGRAM _csp_case_closing_lowest
VAR
END_VAR

;

END_PROGRAM

// ---- Application/CSP/Case/Discharge/_Tasks/_csp_case_discharge_lowest.TcPOU
(*********************************** G.D S.p.A. - Technical Department ***********************************
============= PROGRAM INFO ============
FOLDER:             TBD
MACHINES INVOLVED:  TBD 

============= DESCRIPTION =============
csp main interface program

============= REVISIONS ===============
Date		Version	 	Author      	Description             
----------	-------		------------  	--------------------------------------------
2019/09/27 	0000.00	 	M.Grasso		Creation of the PRG

**********************************************************************************************************)
PROGRAM _csp_case_discharge_lowest
VAR
END_VAR

;

END_PROGRAM

// ---- Application/CSP/Case/Feed/_Tasks/_csp_case_feed_lowest.TcPOU
(*********************************** G.D S.p.A. - Technical Department ***********************************
============= PROGRAM INFO ============
FOLDER:             TBD
MACHINES INVOLVED:  TBD 

============= DESCRIPTION =============
csp main interface program

============= REVISIONS ===============
Date		Version	 	Author      	Description             
----------	-------		------------  	--------------------------------------------
2019/09/27 	0000.00	 	M.Grasso		Creation of the PRG

**********************************************************************************************************)
PROGRAM _csp_case_feed_lowest
VAR
END_VAR

;

END_PROGRAM

// ---- Application/CSP/Case/Flap Control/_Tasks/_csp_case_flapControl_lowest.TcPOU
(*********************************** G.D S.p.A. - Technical Department ***********************************
============= PROGRAM INFO ============
FOLDER:             TBD
MACHINES INVOLVED:  TBD 

============= DESCRIPTION =============
csp main interface program

============= REVISIONS ===============
Date		Version	 	Author      	Description             
----------	-------		------------  	--------------------------------------------
2019/09/27 	0000.00	 	M.Grasso		Creation of the PRG

**********************************************************************************************************)
PROGRAM _csp_case_flapControl_lowest
VAR
END_VAR

;

END_PROGRAM

// ---- Application/CSP/Case/Glue/_Tasks/_csp_case_glue_lowest.TcPOU
(*********************************** G.D S.p.A. - Technical Department ***********************************
============= PROGRAM INFO ============
FOLDER:             TBD
MACHINES INVOLVED:  TBD 

============= DESCRIPTION =============
csp main interface program

============= REVISIONS ===============
Date		Version	 	Author      	Description             
----------	-------		------------  	--------------------------------------------
2019/09/27 	0000.00	 	M.Grasso		Creation of the PRG

**********************************************************************************************************)
PROGRAM _csp_case_glue_lowest
VAR
END_VAR

;

END_PROGRAM

// ---- Application/CSP/Case/Loader/_Tasks/_csp_case_loader_lowest.TcPOU
(*********************************** G.D S.p.A. - Technical Department ***********************************
============= PROGRAM INFO ============
FOLDER:             TBD
MACHINES INVOLVED:  TBD 

============= DESCRIPTION =============
csp main interface program

============= REVISIONS ===============
Date		Version	 	Author      	Description             
----------	-------		------------  	--------------------------------------------
2019/09/27 	0000.00	 	M.Grasso		Creation of the PRG

**********************************************************************************************************)
PROGRAM _csp_case_loader_lowest
VAR
END_VAR

;

END_PROGRAM

// ---- Application/CSP/Case/Open Flap/_Tasks/_csp_case_openFlap_lowest.TcPOU
(*********************************** G.D S.p.A. - Technical Department ***********************************
============= PROGRAM INFO ============
FOLDER:             TBD
MACHINES INVOLVED:  TBD 

============= DESCRIPTION =============
csp main interface program

============= REVISIONS ===============
Date		Version	 	Author      	Description             
----------	-------		------------  	--------------------------------------------
2019/09/27 	0000.00	 	M.Grasso		Creation of the PRG

**********************************************************************************************************)
PROGRAM _csp_case_openFlap_lowest
VAR
END_VAR

;

END_PROGRAM

// ---- Application/CSP/Case/Main/_Tasks/_csp_case_main_lowest.TcPOU
(*********************************** G.D S.p.A. - Technical Department ***********************************
============= PROGRAM INFO ============
FOLDER:             TBD
MACHINES INVOLVED:  TBD 

============= DESCRIPTION =============
csp main interface program

============= REVISIONS ===============
Date		Version	 	Author      	Description             
----------	-------		------------  	--------------------------------------------
2019/09/27 	0000.00	 	M.Grasso		Creation of the PRG

**********************************************************************************************************)
PROGRAM _csp_case_main_lowest
VAR
END_VAR

(*MAIN*)

	(*Brand*)
	
	(*Drives*)
	
	(*Motorization*)
	
	(*Cam Manager*)
	
	(*Services*)
	
	(*Interface*)
	
	(*Safety*)
	
	(* Cabinet *)
	csp_case_main_cabinet()
	;

END_PROGRAM

// ---- Application/CSP/Case/Main/Cabinet/csp_case_main_cabinet.TcPOU
(*********************************** G.D S.p.A. - Technical Department ***********************************
============= PROGRAM INFO ============
FOLDER:             TBD
MACHINES INVOLVED:  TBD 

============= DESCRIPTION =============
csp main program

============= REVISIONS ===============
Date		Version	 	Author      	Description             
----------	-------		------------  	--------------------------------------------
2020/07/08 	0000.00	 	N.Diskin		Creation of the PRG

**********************************************************************************************************)
(*$R
	process_ref := prc;
$*)
PROGRAM csp_case_main_cabinet
VAR
	prc:												process;
	prc_path:											STRING;
	
	temperature_fault_di:								digital_input;
	temperature_fault_dchk:								digital_check;
	
	ups_battery_charge_di:								digital_input;
	ups_battery_mode_di:								digital_input;
	ups_alarm_di:										digital_input;
	
END_VAR

_read_var_input();

_object_manager();

IF NOT objects_running()
THEN
	RETURN;	
END_IF

_read_process_image();

_mode_manager();

CASE process_get_mode(prc) of
	MODE_ABSENT,
	MODE_INACTIVE:
		RETURN;
	MODE_TEST:
		_handle_process_test();
END_CASE

_set_runtime_properties();

(********************************* BODY *********************************)

(************************************************************************)

_handle_messages();

_write_output();

ACTION _handle_messages:
;
END_ACTION

ACTION _handle_process_test:
;
END_ACTION

ACTION _mode_manager:
IF process_mode_req_is_pending(prc)
THEN
    process_apply_mode_req_first_step(prc);
    CASE process_get_mode(prc) OF
        MODE_TO_ABSENT:
			;
        MODE_TO_INACTIVE:
			;
        MODE_TO_TEST:
			;
        MODE_TO_OPERATIONAL:
			;
    END_CASE
    process_apply_mode_req_second_step(prc);
END_IF
END_ACTION

ACTION _object_manager:
IF objects_initialization()
THEN
	sub_process_init(
		object_name					:= 'csp_case_main_cabinet.prc', 
		process						:= csp_case_main.prc, 
		CONVERSION_this				:= prc);
		
	prc_path 						:= process_get_path(prc);
	
	

	digital_input_init(
		object_name					:= CONCAT(prc_path, '_temperature_fault_di'), 
		polarity_direct				:= TRUE, 
		process						:= prc, 
		CONVERSION_this				:= temperature_fault_di);
		
	digital_check_init(
		object_name					:= CONCAT(prc_path, '_temperature_fault_dchk'),
		alarm_if_input_off			:= FALSE,
		alarm_delay					:= 1000,
		enabled_at_powerup			:= TRUE,
		process						:= prc,
		CONVERSION_this				:= temperature_fault_dchk);

	digital_check_add_di(
		di							:= temperature_fault_di,
		CONVERSION_this				:= temperature_fault_dchk);
		
		
	digital_input_init(
		object_name					:= CONCAT(prc_path, '_ups_battery_charge_di'), 
		polarity_direct				:= TRUE, 
		process						:= prc, 
		CONVERSION_this				:= ups_battery_charge_di);
		
	digital_input_init(
		object_name					:= CONCAT(prc_path, '_ups_battery_mode_di'), 
		polarity_direct				:= TRUE, 
		process						:= prc, 
		CONVERSION_this				:= ups_battery_mode_di);
		
	digital_input_init(
		object_name					:= CONCAT(prc_path, '_ups_alarm_di'), 
		polarity_direct				:= TRUE, 
		process						:= prc, 
		CONVERSION_this				:= ups_alarm_di);
	
END_IF

IF objects_running()
THEN
	process_cycle(prc);
	digital_check_cycle(temperature_fault_dchk);
	
END_IF
END_ACTION

ACTION _read_process_image:
;
END_ACTION

ACTION _read_var_input:
;
END_ACTION

ACTION _set_runtime_properties:
;
END_ACTION

ACTION _write_output:
;
END_ACTION

END_PROGRAM

// ---- Application/CSP/Case/Top Rail/_Tasks/_csp_case_topRail_lowest.TcPOU
(*********************************** G.D S.p.A. - Technical Department ***********************************
============= PROGRAM INFO ============
FOLDER:             TBD
MACHINES INVOLVED:  TBD 

============= DESCRIPTION =============
csp main interface program

============= REVISIONS ===============
Date		Version	 	Author      	Description             
----------	-------		------------  	--------------------------------------------
2019/09/27 	0000.00	 	M.Grasso		Creation of the PRG

**********************************************************************************************************)
PROGRAM _csp_case_topRail_lowest
VAR
END_VAR

;

END_PROGRAM

// ---- Application/CSP/Case/Transport/_Tasks/_csp_case_transport_lowest.TcPOU
(*********************************** G.D S.p.A. - Technical Department ***********************************
============= PROGRAM INFO ============
FOLDER:             TBD
MACHINES INVOLVED:  TBD 

============= DESCRIPTION =============
csp main interface program

============= REVISIONS ===============
Date		Version	 	Author      	Description             
----------	-------		------------  	--------------------------------------------
2019/09/27 	0000.00	 	M.Grasso		Creation of the PRG

**********************************************************************************************************)
PROGRAM _csp_case_transport_lowest
VAR
END_VAR

;

END_PROGRAM

// ---- Application/CSP/Transfer/_Tasks/_csp_transfer_lowest.TcPOU
(*********************************** G.D S.p.A. - Technical Department ***********************************
============= PROGRAM INFO ============
FOLDER:             TBD
MACHINES INVOLVED:  TBD 

============= DESCRIPTION =============
csp main interface program

============= REVISIONS ===============
Date		Version	 	Author      	Description             
----------	-------		------------  	--------------------------------------------
2019/09/27 	0000.00	 	M.Grasso		Creation of the PRG

**********************************************************************************************************)
PROGRAM _csp_transfer_lowest
VAR
END_VAR

_csp_transfer_accumulator_lowest();

_csp_transfer_crosspusher_lowest();

_csp_transfer_main_lowest();

_csp_transfer_infeed_lowest();

_csp_transfer_upstacker_lowest();

END_PROGRAM

// ---- Application/CSP/Transfer/Accumulator/_Tasks/_csp_transfer_accumulator_lowest.TcPOU
(*********************************** G.D S.p.A. - Technical Department ***********************************
============= PROGRAM INFO ============
FOLDER:             TBD
MACHINES INVOLVED:  TBD 

============= DESCRIPTION =============
csp main interface program

============= REVISIONS ===============
Date		Version	 	Author      	Description             
----------	-------		------------  	--------------------------------------------
2019/09/27 	0000.00	 	M.Grasso		Creation of the PRG

**********************************************************************************************************)
PROGRAM _csp_transfer_accumulator_lowest
VAR
END_VAR

;

END_PROGRAM

// ---- Application/CSP/Main/_Tasks/_csp_main_lowest.TcPOU
(*********************************** G.D S.p.A. - Technical Department ***********************************
============= PROGRAM INFO ============
FOLDER:             TBD
MACHINES INVOLVED:  TBD 

============= DESCRIPTION =============
csp main interface program

============= REVISIONS ===============
Date		Version	 	Author      	Description             
----------	-------		------------  	--------------------------------------------
2019/09/27 	0000.00	 	M.Grasso		Creation of the PRG

**********************************************************************************************************)
PROGRAM _csp_main_lowest
VAR
END_VAR

(*MAIN*)
	
	(*Drives*)
	
	(*Motorization*)
	
	(*Cam Manager*)
	
	(*Services*)
	
	(*Interface*)
	
	(*Safety*)
	;

END_PROGRAM

// ---- Application/CSP/Customer Interface/_Tasks/_csp_customerInterfaces_lowest.TcPOU
(*********************************** G.D S.p.A. - Technical Department ***********************************
============= PROGRAM INFO ============
FOLDER:             TBD
MACHINES INVOLVED:  TBD 

============= DESCRIPTION =============
Low task

============= REVISIONS ===============
Date		Version	 	Author      	Description             
----------	-------		------------  	--------------------------------------------
2019/03/28 	0000.00	 	CEC 		Creation of the PRG

**********************************************************************************************************)

PROGRAM _csp_customerInterfaces_lowest
VAR
END_VAR

		csp_customerInterfaces();

END_PROGRAM

// ---- Application/_Tasks/_low.TcPOU
(*********************************** G.D S.p.A. - Technical Department ***********************************
============= PROGRAM INFO ============
FOLDER:             TBD
MACHINES INVOLVED:  TBD 

============= DESCRIPTION =============
Low task

============= REVISIONS ===============
Date		Version	 	Author      	Description             
----------	-------		------------  	--------------------------------------------
2019/04/05 	0000.00	 	G.Cera 			Creation of the PRG

**********************************************************************************************************)
{attribute 'TcCallAfterOutputUpdate'}
PROGRAM _low
VAR
END_VAR

(* APPLICATION *)
framework_lowtask_begin();

application_status_manager_low();

_csp_low();

//dbg_low();

framework_lowtask_end();

END_PROGRAM

// ---- Application/_Tasks/Application Status Manager/application_status_manager_low.TcPOU
(********************* G.D S.p.A. - Technical Department ***********************************
Date        Version Author      	Description             
----------  ------- ----------- 	--------------------------------------------------------
2019/04/23	0000.01	G.Cera			Creation of the POU

DESCRIPTION:
Manager of the application status low. it is called by highest speed task


NOTES:

********************************************************************************************)
PROGRAM application_status_manager_low
VAR

END_VAR

VAR_OUTPUT

END_VAR

IF g_application_status=APPLICATION_STATUS_1ST_POWERUP_ABSOLUTE
THEN
   	g_application_status_1st_powerup_low_absolute:=TRUE;
END_IF

IF g_application_status=APPLICATION_STATUS_1ST_POWERUP
THEN
   	g_application_status_1st_powerup_low:=TRUE;
END_IF

IF g_application_status=APPLICATION_STATUS_2ND_POWERUP
THEN
   	g_application_status_2nd_powerup_low:=TRUE;
END_IF

IF g_application_status=APPLICATION_STATUS_3RD_POWERUP
THEN
   	g_application_status_3rd_powerup_low:=TRUE;
END_IF;

END_PROGRAM

// ---- Application/CSP/_Tasks/_csp_low.TcPOU
(*********************************** G.D S.p.A. - Technical Department ***********************************
============= PROGRAM INFO ============
FOLDER:             TBD
MACHINES INVOLVED:  TBD 

============= DESCRIPTION =============
CSP: low task

============= REVISIONS ===============
Date		Version	 	Author      	Description             
----------	-------		------------  	--------------------------------------------
2019/04/05 	0000.00	 	G.Cera 			Creation of the PRG

**********************************************************************************************************)

PROGRAM _csp_low
VAR
END_VAR

_csp_case_low();

_csp_transfer_low();

_csp_main_low();

_csp_customerInterfaces_low();

END_PROGRAM

// ---- Application/CSP/Case/_Tasks/_csp_case_low.TcPOU
(*********************************** G.D S.p.A. - Technical Department ***********************************
============= PROGRAM INFO ============
FOLDER:             TBD
MACHINES INVOLVED:  TBD 

============= DESCRIPTION =============
csp main interface program

============= REVISIONS ===============
Date		Version	 	Author      	Description             
----------	-------		------------  	--------------------------------------------
2019/09/27 	0000.00	 	M.Grasso		Creation of the PRG

**********************************************************************************************************)
PROGRAM _csp_case_low
VAR
END_VAR

_csp_case_closing_low();

_csp_case_discharge_low();

_csp_case_feed_low();

_csp_case_flapControl_low();

_csp_case_glue_low();

_csp_case_loader_low();

_csp_case_openFlap_low();

_csp_case_main_low();

_csp_case_topRail_low();

_csp_case_transport_low();

END_PROGRAM

// ---- Application/CSP/Case/Closing/_Tasks/_csp_case_closing_low.TcPOU
(*********************************** G.D S.p.A. - Technical Department ***********************************
============= PROGRAM INFO ============
FOLDER:             TBD
MACHINES INVOLVED:  TBD 

============= DESCRIPTION =============
csp main interface program

============= REVISIONS ===============
Date		Version	 	Author      	Description             
----------	-------		------------  	--------------------------------------------
2019/09/27 	0000.00	 	M.Grasso		Creation of the PRG

**********************************************************************************************************)
PROGRAM _csp_case_closing_low
VAR
END_VAR

(* CASE *)
	(* CLOSING *)
		(* OS *)
	
		(* LS *)

END_PROGRAM

// ---- Application/CSP/Case/Discharge/_Tasks/_csp_case_discharge_low.TcPOU
(*********************************** G.D S.p.A. - Technical Department ***********************************
============= PROGRAM INFO ============
FOLDER:             TBD
MACHINES INVOLVED:  TBD 

============= DESCRIPTION =============
csp main interface program

============= REVISIONS ===============
Date		Version	 	Author      	Description             
----------	-------		------------  	--------------------------------------------
2019/09/27 	0000.00	 	M.Grasso		Creation of the PRG

**********************************************************************************************************)
PROGRAM _csp_case_discharge_low
VAR
END_VAR

(* CASE *)
	(* DISCHARGE *)
		(* SPEEDBELT *)
		csp_case_discharge_speedBelt_os();
		csp_case_discharge_speedBelt_ls();
		(* SENSORS *)
		;
		(* REJECT *)
		csp_case_discharge_reject_belt();
		csp_case_discharge_reject_modsort();
		csp_case_discharge_reject_sensors();

END_PROGRAM

// ---- Application/CSP/Case/Feed/_Tasks/_csp_case_feed_low.TcPOU
(*********************************** G.D S.p.A. - Technical Department ***********************************
============= PROGRAM INFO ============
FOLDER:             TBD
MACHINES INVOLVED:  TBD 

============= DESCRIPTION =============
csp main interface program

============= REVISIONS ===============
Date		Version	 	Author      	Description             
----------	-------		------------  	--------------------------------------------
2019/09/27 	0000.00	 	M.Grasso		Creation of the PRG

**********************************************************************************************************)
PROGRAM _csp_case_feed_low
VAR
END_VAR

(* CASE *)
	(* FEED *)
		(* ARM *)

		(* MAGAZINE *)
			(* ACC-U-CHANGE *)
			csp_case_feed_magazine_accU();
			csp_case_feed_magazine_accU_osDepth();
			csp_case_feed_magazine_accU_lsDepth();
			(* SENSORS *)
			csp_case_feed_magazine_level();
			csp_case_feed_magazine_level_zone1();
			csp_case_feed_magazine_level_zone2();
			csp_case_feed_magazine_level_zone3();
			csp_case_feed_magazine_level_zone4();
			csp_case_feed_magazine_level_zonelow();
			csp_case_feed_magazine_level_zonemin();
			(* OS *)
			csp_case_feed_magazine_os();
			csp_case_feed_magazine_os_belt();
			csp_case_feed_magazine_os_pusher();
			csp_case_feed_magazine_os_pusherTilt();
			csp_case_feed_magazine_os_sensors();
			(* LS *)
			csp_case_feed_magazine_ls();
			csp_case_feed_magazine_ls_belt();
			csp_case_feed_magazine_ls_pusher();
			csp_case_feed_magazine_ls_pusherTilt();
			csp_case_feed_magazine_ls_sensors();

		(* REJECT *)
			csp_case_feed_reject_belt();
			csp_case_feed_reject_belt_lower();
			csp_case_feed_reject_belt_upper();
			csp_case_feed_reject_sensors();
		(* SHUTTLE *)
			(* ACC-U-CHANGE *)
			csp_case_feed_shuttle_accU();
			csp_case_feed_shuttle_accU_depth();
			csp_case_feed_reject_accU_depth();

END_PROGRAM

// ---- Application/CSP/Case/Flap Control/_Tasks/_csp_case_flapControl_low.TcPOU
(*********************************** G.D S.p.A. - Technical Department ***********************************
============= PROGRAM INFO ============
FOLDER:             TBD
MACHINES INVOLVED:  TBD 

============= DESCRIPTION =============
csp main interface program

============= REVISIONS ===============
Date		Version	 	Author      	Description             
----------	-------		------------  	--------------------------------------------
2019/09/27 	0000.00	 	M.Grasso		Creation of the PRG

**********************************************************************************************************)
PROGRAM _csp_case_flapControl_low
VAR
END_VAR

(* CASE *)
	(* FLAP CONTROL *)
		(* BACKSTOP *)
		;

END_PROGRAM

// ---- Application/CSP/Case/Glue/_Tasks/_csp_case_glue_low.TcPOU
(*********************************** G.D S.p.A. - Technical Department ***********************************
============= PROGRAM INFO ============
FOLDER:             TBD
MACHINES INVOLVED:  TBD 

============= DESCRIPTION =============
csp main interface program

============= REVISIONS ===============
Date		Version	 	Author      	Description             
----------	-------		------------  	--------------------------------------------
2019/09/27 	0000.00	 	M.Grasso		Creation of the PRG

**********************************************************************************************************)
PROGRAM _csp_case_glue_low
VAR
END_VAR

(* CASE *)
	(* GLUE *)
		(* LS *)
			(* ACC-U-CHANGE*)
			csp_case_glue_ls_accU();
			csp_case_glue_ls_accU_lowerPosition();
			csp_case_glue_ls_accU_upperPosition();
		(* OS *)
			(* ACC-U-CHANGE*)
			csp_case_glue_os_accU();
			csp_case_glue_os_accU_lowerPosition();
			csp_case_glue_os_accU_upperPosition();
			csp_case_glue_os_accU_Width();
		(* SENSORS *)
		;

END_PROGRAM

// ---- Application/CSP/Case/Loader/_Tasks/_csp_case_loader_low.TcPOU
(*********************************** G.D S.p.A. - Technical Department ***********************************
============= PROGRAM INFO ============
FOLDER:             TBD
MACHINES INVOLVED:  TBD 

============= DESCRIPTION =============
csp main interface program

============= REVISIONS ===============
Date		Version	 	Author      	Description             
----------	-------		------------  	--------------------------------------------
2019/09/27 	0000.00	 	M.Grasso		Creation of the PRG

**********************************************************************************************************)
PROGRAM _csp_case_loader_low
VAR
END_VAR

(* CASE *)
	(* LOADER *)
		(* GUIDE *)
			(* ACC-U-CHANGE *)
			csp_case_loader_guide_accU();
			csp_case_loader_guide_accU_width();
			(* DOWNSTREAM *)
			csp_case_loader_guide_downstream();
			(* UPSTREAM *)
			csp_case_loader_guide_upstream();
			(* LENGTH *)
			csp_case_loader_guide_length();
		(* PUSHER *)
		;

END_PROGRAM

// ---- Application/CSP/Case/Open Flap/_Tasks/_csp_case_openFlap_low.TcPOU
(*********************************** G.D S.p.A. - Technical Department ***********************************
============= PROGRAM INFO ============
FOLDER:             TBD
MACHINES INVOLVED:  TBD 

============= DESCRIPTION =============
csp main interface program

============= REVISIONS ===============
Date		Version	 	Author      	Description             
----------	-------		------------  	--------------------------------------------
2019/09/27 	0000.00	 	M.Grasso		Creation of the PRG

**********************************************************************************************************)
PROGRAM _csp_case_openFlap_low
VAR
END_VAR

;

END_PROGRAM

// ---- Application/CSP/Case/Main/_Tasks/_csp_case_main_low.TcPOU
(*********************************** G.D S.p.A. - Technical Department ***********************************
============= PROGRAM INFO ============
FOLDER:             TBD
MACHINES INVOLVED:  TBD 

============= DESCRIPTION =============
csp main interface program

============= REVISIONS ===============
Date		Version	 	Author      	Description             
----------	-------		------------  	--------------------------------------------
2019/09/27 	0000.00	 	M.Grasso		Creation of the PRG

**********************************************************************************************************)
PROGRAM _csp_case_main_low
VAR
END_VAR

(*MAIN*)
csp_case_main();

	
	(*Safety*)
	csp_case_main_safety();
	csp_case_main_safety_token();
		csp_case_main_safety_guards();
	
		csp_case_main_safety_emergency();

		csp_case_main_safety_drives();
			csp_case_main_safety_drives_commonConfiguration();
			csp_case_main_safety_accUChange();
			csp_case_main_safety_conveyor();
			csp_case_main_safety_air();
			csp_case_main_safety_drives_PS2000(); 
			csp_case_main_safety_drives_SD2100(); 
			csp_case_main_safety_drives_SD2200(); 
			csp_case_main_safety_drives_SD2300(); 
			csp_case_main_safety_drives_SD2400(); 
			csp_case_main_safety_drives_SD2500(); 
			csp_case_main_safety_drives_SD12000(); 
			csp_case_main_safety_drives_SD8000(); 
			csp_case_main_safety_drives_SD8100(); 
			csp_case_main_safety_drives_SD8200(); 
			csp_case_main_safety_drives_SD8300(); 
			csp_case_main_safety_drives_SD8400(); 
			csp_case_main_safety_drives_SD8500(); 
			csp_case_main_safety_drives_SD8600(); 
			csp_case_main_safety_drives_SD10000(); 
			csp_case_main_safety_drives_SD10100(); 
			csp_case_main_safety_drives_SD10200(); 
			csp_case_main_safety_drives_SD10300(); 
			csp_case_main_safety_drives_SD10400(); 
			csp_case_main_safety_drives_SD11000(); 
			csp_case_main_safety_drives_SD15000();  
			csp_case_main_safety_drives_SD26000();
			csp_case_main_safety_drives_SD26100(); 
		
		csp_case_main_safety_interface(); 
		
		csp_case_main_cabinet_sync_unit(
				parent_prc 				:= csp_case_main_cabinet.prc,
				cabinet_ethercat_master := csp_main.cabinet_ethercat_master);

END_PROGRAM

// ---- Application/CSP/Case/Main/Safety/csp_case_main_safety.TcPOU
(*********************************** G.D S.p.A. - Technical Department ***********************************
============= PROGRAM INFO ============
FOLDER:             TBD
MACHINES INVOLVED:  TBD 

============= DESCRIPTION =============

============= REVISIONS ===============
Date		Version	 	Author      	Description             
----------	-------		------------  	--------------------------------------------
2019/04/24 	0000.00	 	M.Grasso		Creation of the PRG

**********************************************************************************************************)
(*$R
	process_ref := prc;
$*)
PROGRAM csp_case_main_safety
VAR
	prc:					process;
	prc_path:				STRING;
	
	series_closed_dvr:		BOOL;
END_VAR

_read_var_input();

_object_manager();

IF NOT objects_running()
THEN
	RETURN;	
END_IF

_read_process_image();

_mode_manager();

CASE process_get_mode(prc) of
	MODE_ABSENT,
	MODE_INACTIVE:
		RETURN;
	MODE_TEST:
		_handle_process_test();
END_CASE

_set_runtime_properties();

(********************************* BODY *********************************)

(************************************************************************)

_handle_messages();

_write_output();

ACTION _handle_messages:
;
END_ACTION

ACTION _handle_process_test:
;
END_ACTION

ACTION _mode_manager:
IF process_mode_req_is_pending(prc)
THEN
    process_apply_mode_req_first_step(prc);
    CASE process_get_mode(prc) OF
        MODE_TO_ABSENT:
			;
        MODE_TO_INACTIVE:
			;
        MODE_TO_TEST:
			;
        MODE_TO_OPERATIONAL:
			;
    END_CASE
    process_apply_mode_req_second_step(prc);
END_IF
END_ACTION

ACTION _object_manager:
IF objects_initialization()
THEN
	sub_process_init(
		object_name					:= 'csp_case_main_safety.prc', 
		process						:= csp_case_main.prc, 
		CONVERSION_this				:= prc);
		
	prc_path 						:= process_get_path(prc);
END_IF

IF objects_running()
THEN
	process_cycle(prc);
END_IF
END_ACTION

ACTION _read_process_image:
series_closed_dvr := 
						(* LIST ALL CASE SIS *)
						csp_case_main_safety_drives_PS2000.safety_integrated_series_close_dvr
					(*	AND
						csp_case_main_safety_drives_sd10000.safety_integrated_series_close_dvr_chA
						AND
						csp_case_main_safety_drives_sd10000.safety_integrated_series_close_dvr_chB
						AND
						csp_case_main_safety_drives_sd10100.safety_integrated_series_close_dvr_chA
						AND
						csp_case_main_safety_drives_sd10100.safety_integrated_series_close_dvr_chB
						AND
						csp_case_main_safety_drives_sd10200.safety_integrated_series_close_dvr_chA
						AND
						csp_case_main_safety_drives_sd10200.safety_integrated_series_close_dvr_chB
						AND
						csp_case_main_safety_drives_sd10300.safety_integrated_series_close_dvr_chA
						AND
						csp_case_main_safety_drives_sd10300.safety_integrated_series_close_dvr_chB
						AND
						csp_case_main_safety_drives_sd10400.safety_integrated_series_close_dvr_chA
						AND
						csp_case_main_safety_drives_sd10400.safety_integrated_series_close_dvr_chB						
						AND
						csp_case_main_safety_drives_sd11000.safety_integrated_series_close_dvr_chA
						//AND
						//safety_integrated_series_is_safely_closed(csp_case_main_safety_drives_sd11000.chB_smes_sis)						
						AND
						csp_case_main_safety_drives_sd12000.safety_integrated_series_close_dvr_chA
						AND
						csp_case_main_safety_drives_sd12000.safety_integrated_series_close_dvr_chB	
						AND
						csp_case_main_safety_drives_sd15000.safety_integrated_series_close_dvr_chA
						AND
						csp_case_main_safety_drives_sd15000.safety_integrated_series_close_dvr_chB*)
						AND
						csp_case_main_safety_drives_sd2100.safety_integrated_series_close_dvr_chA
						AND
						csp_case_main_safety_drives_sd2100.safety_integrated_series_close_dvr_chB
						AND
						csp_case_main_safety_drives_sd2200.safety_integrated_series_close_dvr_chA
						AND
						csp_case_main_safety_drives_sd2200.safety_integrated_series_close_dvr_chB
						(*AND
						csp_case_main_safety_drives_sd2300.safety_integrated_series_close_dvr_chA
						AND
						csp_case_main_safety_drives_sd2300.safety_integrated_series_close_dvr_chB
						AND
						csp_case_main_safety_drives_sd2400.safety_integrated_series_close_dvr_chA
						AND
						csp_case_main_safety_drives_sd2400.safety_integrated_series_close_dvr_chB						
						AND
						csp_case_main_safety_drives_sd2500.safety_integrated_series_close_dvr_chA
						AND
						csp_case_main_safety_drives_sd2500.safety_integrated_series_close_dvr_chB
						AND
						csp_case_main_safety_drives_sd26000.safety_integrated_series_close_dvr_chA
						AND
						csp_case_main_safety_drives_sd26000.safety_integrated_series_close_dvr_chB					
						AND
						csp_case_main_safety_drives_sd26100.safety_integrated_series_close_dvr_chA
						AND
						csp_case_main_safety_drives_sd26100.safety_integrated_series_close_dvr_chB
						AND
						csp_case_main_safety_drives_sd8000.safety_integrated_series_close_dvr_chA
						AND
						csp_case_main_safety_drives_sd8000.safety_integrated_series_close_dvr_chB					
						AND
						csp_case_main_safety_drives_sd8100.safety_integrated_series_close_dvr_chA
						AND
						csp_case_main_safety_drives_sd8100.safety_integrated_series_close_dvr_chB		
						AND
						csp_case_main_safety_drives_sd8200.safety_integrated_series_close_dvr_chA
						AND
						csp_case_main_safety_drives_sd8200.safety_integrated_series_close_dvr_chB		
						AND
						csp_case_main_safety_drives_sd8300.safety_integrated_series_close_dvr_chA
						AND
						csp_case_main_safety_drives_sd8300.safety_integrated_series_close_dvr_chB		
						AND
						csp_case_main_safety_drives_sd8400.safety_integrated_series_close_dvr_chA
						AND
						csp_case_main_safety_drives_sd8400.safety_integrated_series_close_dvr_chB		
						AND
						csp_case_main_safety_drives_sd8500.safety_integrated_series_close_dvr_chA
						AND
						csp_case_main_safety_drives_sd8500.safety_integrated_series_close_dvr_chB	
						AND
						csp_case_main_safety_drives_sd8600.safety_integrated_series_close_dvr_chA
						AND
						csp_case_main_safety_drives_sd8600.safety_integrated_series_close_dvr_chB	*)			
;
END_ACTION

ACTION _read_var_input:
;
END_ACTION

ACTION _set_runtime_properties:
;
END_ACTION

ACTION _write_output:
;
END_ACTION

END_PROGRAM

// ---- Application/CSP/Case/Top Rail/_Tasks/_csp_case_topRail_low.TcPOU
(*********************************** G.D S.p.A. - Technical Department ***********************************
============= PROGRAM INFO ============
FOLDER:             TBD
MACHINES INVOLVED:  TBD 

============= DESCRIPTION =============
csp main interface program

============= REVISIONS ===============
Date		Version	 	Author      	Description             
----------	-------		------------  	--------------------------------------------
2019/09/27 	0000.00	 	M.Grasso		Creation of the PRG

**********************************************************************************************************)
PROGRAM _csp_case_topRail_low
VAR
END_VAR

(* CASE *)
	(* TOP RAIL *)
		(* ACC-U-CHANGE *)
			(* LS *)
			csp_case_tr_accU_ls();
			csp_case_tr_accU_ls_width();
			(* OS *)
			csp_case_tr_accU_Os();
			csp_case_tr_accU_Os_width();
			(* DEPTH *)
			csp_case_tr_accU_depth();
			(* VIRTUAL MASTER *)
			csp_case_tr_accU_virtualMaster();
			
		(* SQUARING *)
			(* LS *)
			csp_case_tr_squaring_ls();
			csp_case_tr_squaring_ls_leading();
			csp_case_tr_squaring_ls_trailing();
			(* OS *)
			csp_case_tr_squaring_os();
			csp_case_tr_squaring_os_leading();
			csp_case_tr_squaring_os_trailing();

END_PROGRAM

// ---- Application/CSP/Case/Transport/_Tasks/_csp_case_transport_low.TcPOU
(*********************************** G.D S.p.A. - Technical Department ***********************************
============= PROGRAM INFO ============
FOLDER:             TBD
MACHINES INVOLVED:  TBD 

============= DESCRIPTION =============
csp main interface program

============= REVISIONS ===============
Date		Version	 	Author      	Description             
----------	-------		------------  	--------------------------------------------
2019/09/27 	0000.00	 	M.Grasso		Creation of the PRG

**********************************************************************************************************)
PROGRAM _csp_case_transport_low
VAR
END_VAR

(* CSP *)
	(* TRANSPORT *)
		(* ACC-U-CHANGE *)
		csp_case_transport_accU_depth();
		csp_case_transport_accU_virtualMaster();
		(* LS *)
		(* OS *)
		csp_case_transport_os_minorPlow();
		(* TENSIONER *)
		;

END_PROGRAM

// ---- Application/CSP/Transfer/_Tasks/_csp_transfer_low.TcPOU
(*********************************** G.D S.p.A. - Technical Department ***********************************
============= PROGRAM INFO ============
FOLDER:             TBD
MACHINES INVOLVED:  TBD 

============= DESCRIPTION =============
csp main interface program

============= REVISIONS ===============
Date		Version	 	Author      	Description             
----------	-------		------------  	--------------------------------------------
2019/09/27 	0000.00	 	M.Grasso		Creation of the PRG

**********************************************************************************************************)
PROGRAM _csp_transfer_low
VAR
END_VAR

_csp_transfer_accumulator_low();

_csp_transfer_crosspusher_low();

_csp_transfer_main_low();

_csp_transfer_infeed_low();

_csp_transfer_upstacker_low();

END_PROGRAM

// ---- Application/CSP/Transfer/Accumulator/_Tasks/_csp_transfer_accumulator_low.TcPOU
(*********************************** G.D S.p.A. - Technical Department ***********************************
============= PROGRAM INFO ============
FOLDER:             TBD
MACHINES INVOLVED:  TBD 

============= DESCRIPTION =============
csp main interface program

============= REVISIONS ===============
Date		Version	 	Author      	Description             
----------	-------		------------  	--------------------------------------------
2019/09/27 	0000.00	 	M.Grasso		Creation of the PRG

**********************************************************************************************************)
PROGRAM _csp_transfer_accumulator_low
VAR
END_VAR

(* TRANSFER *)
	(* ACCUMULATOR *)
		(* ACCU-U-CHANGE*)
			(* TOP RAIL LENGTH *)
			csp_transfer_accumulator_accU_topRailLength();
			(* TOP RAIL WIDTH *)
			csp_transfer_accumulator_accU_topRailWidth();
			(* DEPTH *)
			csp_transfer_accumulator_accU_depth();
			(* CONVEYOR DEPTH*)
			csp_transfer_accumulator_accU_convDepth();
			
			csp_transfer_accumulator_accU_virtualMaster();
			
		(* FINGER *)
			(* LS *)
			csp_transfer_accumulator_finger_ls();
			(* OS *)
			csp_transfer_accumulator_finger_os();
		(* LIFT *)
		;

END_PROGRAM

// ---- Application/CSP/Main/_Tasks/_csp_main_low.TcPOU
(*********************************** G.D S.p.A. - Technical Department ***********************************
============= PROGRAM INFO ============
FOLDER:             TBD
MACHINES INVOLVED:  TBD 

============= DESCRIPTION =============
csp main interface program

============= REVISIONS ===============
Date		Version	 	Author      	Description             
----------	-------		------------  	--------------------------------------------
2019/09/27 	0000.00	 	M.Grasso		Creation of the PRG

**********************************************************************************************************)
PROGRAM _csp_main_low
VAR
END_VAR

(*MAIN*)
csp_main();

	(*Brand*)
	csp_main_brand();
	(*Drives*)
	
	(*Motorization*)
	csp_main_motorization();
	(*Cam Manager*)
	
	(*Services*)
	csp_main_productionData();
	(*Interface*)
	csp_main_interface_cabinet();
	(*Safety*)
	csp_main_safety();
	csp_main_safety_interface();
	csp_main_safety_connectionShutDown();
	csp_main_safety_drives();
		//csp_main_safety_drives_powerSupply();
	(*Jog Manager*)
	csp_main_jogManager();

END_PROGRAM

// ---- Application/CSP/Main/Production Data/csp_main_productionData.TcPOU
(*********************************** G.D S.p.A. - Technical Department ***********************************
============= PROGRAM INFO ============
FOLDER:             TBD
MACHINES INVOLVED:  TBD 

============= DESCRIPTION =============
Production data management

============= REVISIONS ===============
Date		Version	 	Author      	Description             
----------	-------		------------  	--------------------------------------------
2020/02/07 	0000.00	 	Gavagni			Creation of the PRG

**********************************************************************************************************)
(*$R process_ref:= prc; $*)

PROGRAM csp_main_productionData
VAR	
	prc:												process;
	prc_path:											STRING;

	reject_reason_code:									reject_reasons_enum;		(*$M $*)
	aux_reason_code:									auxiliary_counters_code_enum; (*$M $*)

END_VAR

_read_var_input();

_object_manager();

IF NOT objects_running()
THEN
	RETURN;	
END_IF

_read_process_image();

_mode_manager();

CASE process_get_mode(prc) OF
	MODE_ABSENT,
	MODE_INACTIVE:
		RETURN;
	MODE_TEST:
		;
END_CASE

_set_runtime_properties();

(********************************* BODY *********************************)

(************************************************************************)

_handle_messages();
_write_output();

ACTION _handle_messages:
;
END_ACTION

ACTION _handle_process_test:
;
END_ACTION

ACTION _mode_manager:
IF process_mode_req_is_pending(prc)
THEN
    process_apply_mode_req_first_step(prc);
    CASE process_get_mode(prc) OF
        MODE_TO_ABSENT:
			;
        MODE_TO_INACTIVE:
			;
        MODE_TO_TEST:
			;
        MODE_TO_OPERATIONAL:
			;
    END_CASE
    process_apply_mode_req_second_step(prc);
END_IF
END_ACTION

ACTION _object_manager:
IF objects_initialization()
THEN
	sub_process_init(
		object_name					:= 'csp_main_productionData.prc', 
		process						:= csp_main.prc, 
		CONVERSION_this				:= prc);
		
	prc_path 						:= process_get_path(prc);
		
END_IF

IF objects_running()
THEN
	process_cycle(prc);
	

END_IF
END_ACTION

ACTION _read_process_image:
;
END_ACTION

ACTION _read_var_input:
;
END_ACTION

ACTION _set_runtime_properties:
;
END_ACTION

ACTION _write_output:
;
END_ACTION

END_PROGRAM

// ---- Application/CSP/Main/Interface/Cabinet/csp_main_interface_cabinet.TcPOU
(*********************************** G.D S.p.A. - Technical Department ***********************************
============= PROGRAM INFO ============
FOLDER:             TBD
MACHINES INVOLVED:  TBD 

============= DESCRIPTION =============
csp - Cabinet interface

============= REVISIONS ===============
Date		Version	 	Author      	Description             
----------	-------		------------  	--------------------------------------------
2019/04/05 	0000.00	 	M.Grasso		Creation of the PRG

**********************************************************************************************************)
(*$R
	process_ref := prc;
$*)
PROGRAM csp_main_interface_cabinet
VAR
	prc:					process;
	prc_path:				STRING;
	
	stop_from_cabinet_asm:	message;
END_VAR

_read_var_input();

_object_manager();

IF NOT objects_running()
THEN
	RETURN;	
END_IF

_read_process_image();

_mode_manager();

CASE process_get_mode(prc) OF
	MODE_ABSENT,
	MODE_INACTIVE:
		RETURN;
	MODE_TEST:
		_handle_process_test();
END_CASE

_set_runtime_properties();

(********************************* BODY *********************************)

(************************************************************************)

_handle_messages();

_write_output();

ACTION _handle_messages:
IF	csp_main.i_cabinet_is_running
THEN
	process_message_reset(stop_from_cabinet_asm);
END_IF
END_ACTION

ACTION _handle_process_test:
;
END_ACTION

ACTION _mode_manager:
IF process_mode_req_is_pending(prc)
THEN
    process_apply_mode_req_first_step(prc);
    CASE process_get_mode(prc) OF
        MODE_TO_ABSENT:
			;
        MODE_TO_INACTIVE:
			;
        MODE_TO_TEST:
			;
        MODE_TO_OPERATIONAL:
			;
    END_CASE
    process_apply_mode_req_second_step(prc);
END_IF
END_ACTION

ACTION _object_manager:
IF objects_initialization()
THEN
	sub_process_init(
		object_name					:= 'csp_main_interface_cabinet.prc', 
		process						:= csp_main_interface.prc, 
		CONVERSION_this				:= prc);
		
	prc_path 						:= process_get_path(prc);
	
	process_message_init(
		object_name					:=	CONCAT(prc_path, '_stop_from_cabinet_asm'),
        behaviour					:=	MESSAGE_BEHAVIOUR_STATE,
		reset_timeout				:=	0,
        disableable					:=	FALSE,
        individual_reset			:=	FALSE,
        machine_reaction			:=	MACHINE_REACTION_NORMAL_STOP,
        typology					:=	MESSAGE_TYPOLOGY_ABNORMAL,
		process						:=	prc,
		CONVERSION_this				:=	stop_from_cabinet_asm);
END_IF

IF objects_running()
THEN
	process_cycle(prc);
END_IF
END_ACTION

ACTION _read_process_image:
;
END_ACTION

ACTION _read_var_input:
;
END_ACTION

ACTION _set_runtime_properties:
;
END_ACTION

ACTION _write_output:
;
END_ACTION

END_PROGRAM

// ---- Application/CSP/Main/Safety/csp_main_safety.TcPOU
(*********************************** G.D S.p.A. - Technical Department ***********************************
============= PROGRAM INFO ============
FOLDER:             TBD
MACHINES INVOLVED:  TBD 

============= DESCRIPTION =============

============= REVISIONS ===============
Date		Version	 	Author      	Description             
----------	-------		------------  	--------------------------------------------
2019/04/24 	0000.00	 	M.Grasso		Creation of the PRG

**********************************************************************************************************)
(*$R
	process_ref := prc;
$*)
PROGRAM csp_main_safety
VAR
	prc:					process;
	prc_path:				STRING;
	
	series_closed_dvr:		BOOL;
	
END_VAR

_read_var_input();

_object_manager();

IF NOT objects_running()
THEN
	RETURN;	
END_IF

_read_process_image();

_mode_manager();

CASE process_get_mode(prc) of
	MODE_ABSENT,
	MODE_INACTIVE:
		RETURN;
	MODE_TEST:
		_handle_process_test();
END_CASE

_set_runtime_properties();

(********************************* BODY *********************************)

(************************************************************************)

_handle_messages();

_write_output();

ACTION _handle_messages:
;
END_ACTION

ACTION _handle_process_test:
;
END_ACTION

ACTION _mode_manager:
IF process_mode_req_is_pending(prc)
THEN
    process_apply_mode_req_first_step(prc);
    CASE process_get_mode(prc) OF
        MODE_TO_ABSENT:
			;
        MODE_TO_INACTIVE:
			;
        MODE_TO_TEST:
			;
        MODE_TO_OPERATIONAL:
			;
    END_CASE
    process_apply_mode_req_second_step(prc);
END_IF
END_ACTION

ACTION _object_manager:
IF objects_initialization()
THEN
	sub_process_init(
		object_name					:= 'csp_main_safety.prc', 
		process						:= csp_main.prc, 
		CONVERSION_this				:= prc);
		
	prc_path 						:= process_get_path(prc);
END_IF

IF objects_running()
THEN
	process_cycle(prc);
END_IF
END_ACTION

ACTION _read_process_image:
	series_closed_dvr := csp_case_main_safety.series_closed_dvr;
END_ACTION

ACTION _read_var_input:
;
END_ACTION

ACTION _set_runtime_properties:
;
END_ACTION

ACTION _write_output:
;
END_ACTION

END_PROGRAM

// ---- Application/CSP/Main/Safety/Interface/csp_main_safety_interface.TcPOU
(*********************************** G.D S.p.A. - Technical Department ***********************************
============= PROGRAM INFO ============
FOLDER:             TBD
MACHINES INVOLVED:  TBD 

============= DESCRIPTION =============
csp machine safety interfaces definition

============= REVISIONS ===============
Date		Version	 	Author      	Description             
----------	-------		------------  	--------------------------------------------
2019/04/24 	0000.00	 	M.Grasso		Creation of the PRG

**********************************************************************************************************)
(*$R
	process_ref := prc;
$*)
PROGRAM csp_main_safety_interface
VAR
	prc:						process;
	prc_path:					STRING;
		
END_VAR

_read_var_input();

_object_manager();

IF NOT objects_running()
THEN
	RETURN;	
END_IF

_read_process_image();

_mode_manager();

CASE process_get_mode(prc) of
	MODE_ABSENT,
	MODE_INACTIVE:
		RETURN;
	MODE_TEST:
		_handle_process_test();
END_CASE

_set_runtime_properties();

(********************************* BODY *********************************)

(************************************************************************)

_handle_messages();

_write_output();

ACTION _handle_messages:
;
END_ACTION

ACTION _handle_process_test:
;
END_ACTION

ACTION _mode_manager:
IF process_mode_req_is_pending(prc)
THEN
    process_apply_mode_req_first_step(prc);
    CASE process_get_mode(prc) OF
        MODE_TO_ABSENT:
			;
        MODE_TO_INACTIVE:
			;
        MODE_TO_TEST:
			;
        MODE_TO_OPERATIONAL:
			;
    END_CASE
    process_apply_mode_req_second_step(prc);
END_IF
END_ACTION

ACTION _object_manager:
IF objects_initialization()
THEN
	sub_process_init(
		object_name								:= 'csp_main_safety_interface.prc', 
		process									:= csp_main_safety.prc, 
		CONVERSION_this							:= prc);
		
	prc_path 									:= process_get_path(prc);
	
END_IF

IF objects_running()
THEN
	process_cycle(prc);
END_IF
END_ACTION

ACTION _read_process_image:
;
END_ACTION

ACTION _read_var_input:
;
END_ACTION

ACTION _set_runtime_properties:
;
END_ACTION

ACTION _write_output:
;
END_ACTION

END_PROGRAM

// ---- Application/CSP/Main/Safety/csp_main_safety_connectionShutDown.TcPOU
(*********************************** G.D S.p.A. - Technical Department ***********************************
============= PROGRAM INFO ============
FOLDER:             TBD
MACHINES INVOLVED:  TBD 

============= DESCRIPTION =============

============= REVISIONS ===============
Date		Version	 	Author      	Description             
----------	-------		------------  	--------------------------------------------
2019/04/24 	0000.00	 	M.Grasso		Creation of the PRG

**********************************************************************************************************)
(*$R
	process_ref := prc;
$*)
PROGRAM csp_main_safety_connectionShutDown
VAR
	prc:												process;
	prc_path:											STRING;
	
	SPLC5000_connectionShutdown_sig:					safety_integrated_group;
	SPLC40210_connectionShutdown_sig:					safety_integrated_group;

END_VAR

_read_var_input();

_object_manager();

IF NOT objects_running()
THEN
	RETURN;	
END_IF

_read_process_image();

_mode_manager();

CASE process_get_mode(prc) of
	MODE_ABSENT,
	MODE_INACTIVE:
		RETURN;
	MODE_TEST:
		_handle_process_test();
END_CASE

_set_runtime_properties();

(********************************* BODY *********************************)

(************************************************************************)

_handle_messages();

_write_output();

ACTION _handle_messages:
;
END_ACTION

ACTION _handle_process_test:
;
END_ACTION

ACTION _mode_manager:
IF process_mode_req_is_pending(prc)
THEN
    process_apply_mode_req_first_step(prc);
    CASE process_get_mode(prc) OF
        MODE_TO_ABSENT:
			;
        MODE_TO_INACTIVE:
			;
        MODE_TO_TEST:
			;
        MODE_TO_OPERATIONAL:
			;
    END_CASE
    process_apply_mode_req_second_step(prc);
END_IF
END_ACTION

ACTION _object_manager:
IF objects_initialization()
THEN
	sub_process_init(
		object_name								:= 'csp_main_safety_connectionShutDown.prc', 
		process									:= csp_main_safety.prc, 
		CONVERSION_this							:= prc);
		
	prc_path 									:= process_get_path(prc);
	
	safety_integrated_group_init(
		object_name								:=	CONCAT(prc_path, '_SPLC5000_connectionShutdown_sig'), 
		controller								:=	csp_case_main_safety_interface.SPLC5000_sic,
		process									:=	prc,
		CONVERSION_this							:=	SPLC5000_connectionShutdown_sig);

END_IF

IF objects_running()
THEN
	process_cycle(prc);
	
	safety_integrated_group_cycle(SPLC5000_connectionShutdown_sig);
END_IF
END_ACTION

ACTION _read_process_image:
;
END_ACTION

ACTION _read_var_input:
;
END_ACTION

ACTION _set_runtime_properties:
;
END_ACTION

ACTION _write_output:
;
END_ACTION

END_PROGRAM

// ---- Application/CSP/Main/Safety/Drives/csp_main_safety_drives.TcPOU

(*********************************** G.D S.p.A. - Technical Department ***********************************
============= PROGRAM INFO ============
FOLDER:             TBD
MACHINES INVOLVED:  TBD 

============= DESCRIPTION =============

============= REVISIONS ===============
Date		Version	 	Author      	Description             
----------	-------		------------  	--------------------------------------------
2019/04/24 	0000.00	 	M.Grasso		Creation of the PRG

**********************************************************************************************************)
(*$R 
	process_ref:= prc; 
$*)
PROGRAM csp_main_safety_drives
VAR
	prc:					process;
	prc_path:				STRING;	
END_VAR

_read_var_input();

_objects_manager();

IF NOT objects_running()
THEN
	RETURN;	
END_IF

_read_process_image();

_mode_manager();

CASE process_get_mode(prc) OF
	MODE_ABSENT,
	MODE_INACTIVE:
		RETURN;
	MODE_TEST:
		;
END_CASE

_set_runtime_properties();

(********************************* BODY *********************************)

(************************************************************************)

_handle_messages();

_write_output();

ACTION _handle_messages:
;
END_ACTION

ACTION _handle_process_test:
;
END_ACTION

ACTION _mode_manager:
IF process_mode_req_is_pending(prc)
THEN
    process_apply_mode_req_first_step(prc);
    CASE process_get_mode(prc) OF
        MODE_TO_ABSENT:
			;
        MODE_TO_INACTIVE:
			;
        MODE_TO_TEST:
			;
        MODE_TO_OPERATIONAL:
			;
    END_CASE
    process_apply_mode_req_second_step(prc);
END_IF
END_ACTION

ACTION _objects_manager:
IF objects_initialization()
THEN
	sub_process_init(
		object_name					:= 'csp_main_safety_drives.prc', 
		process						:= csp_main_safety.prc, 
		CONVERSION_this				:= prc);
		
	prc_path 						:= process_get_path(prc);		
END_IF

IF objects_running()
THEN
	process_cycle(prc);
END_IF
END_ACTION

ACTION _read_process_image:
;
END_ACTION

ACTION _read_var_input:
;
END_ACTION

ACTION _set_runtime_properties:
;
END_ACTION

ACTION _write_output:
;
END_ACTION

END_PROGRAM

// ---- Application/CSP/Customer Interface/_Tasks/_csp_customerInterfaces_low.TcPOU
(*********************************** G.D S.p.A. - Technical Department ***********************************
============= PROGRAM INFO ============
FOLDER:             TBD
MACHINES INVOLVED:  TBD 

============= DESCRIPTION =============
Low task

============= REVISIONS ===============
Date		Version	 	Author      	Description             
----------	-------		------------  	--------------------------------------------
2019/03/28 	0000.00	 	CEC 			Creation of the PRG

**********************************************************************************************************)

PROGRAM _csp_customerInterfaces_low
VAR
END_VAR

;

END_PROGRAM

// ---- Application/_Tasks/_normal.TcPOU
(*********************************** G.D S.p.A. - Technical Department ***********************************
============= PROGRAM INFO ============
FOLDER:             TBD
MACHINES INVOLVED:  TBD 

============= DESCRIPTION =============
Highest task

============= REVISIONS ===============
Date		Version	 	Author      	Description             
----------	-------		------------  	--------------------------------------------
2019/04/05 	0000.00	 	G.Cera 			Creation of the PRG

**********************************************************************************************************)
{attribute 'TcCallAfterOutputUpdate'}
PROGRAM _normal
VAR
END_VAR

(* APPLICATION *)
framework_normaltask_begin();
application_status_manager();
application_status_manager_normal();

_csp_normal();

//dbg_normal();

framework_normaltask_end();

END_PROGRAM

// ---- Application/_Tasks/Application Status Manager/application_status_manager.TcPOU
(********************* G.D S.p.A. - Technical Department ***********************************
Date        Version Author      	Description             
----------  ------- ----------- 	--------------------------------------------------------
2019/04/23	0000.01	G.Cera			Creation of the POU

DESCRIPTION:
Manager of the application status. it is called by highest speed task

NOTES:

********************************************************************************************)
PROGRAM application_status_manager
VAR

END_VAR

VAR_OUTPUT

END_VAR

IF NOT objects_running()
THEN
	g_application_status					:=	APPLICATION_STATUS_NOT_INITIALIZED;

	g_application_status_1st_powerup_high	:=	FALSE;
	g_application_status_1st_powerup_normal	:=	FALSE;
	g_application_status_1st_powerup_low	:=	FALSE;

	g_application_status_2nd_powerup_high	:=	FALSE;
	g_application_status_2nd_powerup_normal	:=	FALSE;
	g_application_status_2nd_powerup_low	:=	FALSE;

	g_application_status_3rd_powerup_high	:=	FALSE;
	g_application_status_3rd_powerup_normal	:=	FALSE;
	g_application_status_3rd_powerup_low	:=	FALSE;

	RETURN;
END_IF

IF	g_application_status=APPLICATION_STATUS_NOT_INITIALIZED
	AND
	(
		NOT g_application_status_1st_powerup_high_absolute
		OR
		NOT g_application_status_1st_powerup_normal_absolute
		OR
		NOT g_application_status_1st_powerup_low_absolute
	)
THEN
	g_application_status					:=	APPLICATION_STATUS_1ST_POWERUP_ABSOLUTE;
END_IF

IF	(
		g_application_status=APPLICATION_STATUS_1ST_POWERUP_ABSOLUTE
		OR
		g_application_status=APPLICATION_STATUS_NOT_INITIALIZED
	)
	AND
	g_application_status_1st_powerup_high_absolute
	AND
	g_application_status_1st_powerup_normal_absolute
	AND
	g_application_status_1st_powerup_low_absolute
THEN
	g_application_status					:=	APPLICATION_STATUS_1ST_POWERUP;
END_IF

IF	g_application_status=APPLICATION_STATUS_1ST_POWERUP
	AND
	g_application_status_1st_powerup_high
	AND
	g_application_status_1st_powerup_normal
	AND
	g_application_status_1st_powerup_low
THEN
	g_application_status					:=	APPLICATION_STATUS_2ND_POWERUP;
END_IF

IF	g_application_status=APPLICATION_STATUS_2ND_POWERUP
	AND
	g_application_status_2nd_powerup_high
	AND
	g_application_status_2nd_powerup_normal
	AND
	g_application_status_2nd_powerup_low
THEN
	g_application_status					:=	APPLICATION_STATUS_3RD_POWERUP;
END_IF

IF	g_application_status=APPLICATION_STATUS_3RD_POWERUP
	AND
	g_application_status_3rd_powerup_high
	AND
	g_application_status_3rd_powerup_normal
	AND
	g_application_status_3rd_powerup_low
THEN
	g_application_status					:=	APPLICATION_STATUS_RUNNING;
END_IF

END_PROGRAM

// ---- Application/_Tasks/Application Status Manager/application_status_manager_normal.TcPOU
(********************* G.D S.p.A. - Technical Department ***********************************
Date        Version Author      	Description             
----------  ------- ----------- 	--------------------------------------------------------
2019/04/23	0000.01	G.Cera			Creation of the POU

DESCRIPTION:
Manager of the application status normal. it is called by highest speed task


NOTES:

********************************************************************************************)
PROGRAM application_status_manager_normal
VAR

END_VAR

VAR_OUTPUT

END_VAR

IF g_application_status=APPLICATION_STATUS_1ST_POWERUP_ABSOLUTE
THEN
   	g_application_status_1st_powerup_normal_absolute:=TRUE;
END_IF

IF g_application_status=APPLICATION_STATUS_1ST_POWERUP
THEN
   	g_application_status_1st_powerup_normal:=TRUE;
END_IF

IF g_application_status=APPLICATION_STATUS_2ND_POWERUP
THEN
   	g_application_status_2nd_powerup_normal:=TRUE;
END_IF

IF g_application_status=APPLICATION_STATUS_3RD_POWERUP
THEN
   	g_application_status_3rd_powerup_normal:=TRUE;
END_IF;

END_PROGRAM

// ---- Application/CSP/_Tasks/_csp_normal.TcPOU
(*********************************** G.D S.p.A. - Technical Department ***********************************
============= PROGRAM INFO ============
FOLDER:             TBD
MACHINES INVOLVED:  TBD 

============= DESCRIPTION =============
CSP: normal task

============= REVISIONS ===============
Date		Version	 	Author      	Description             
----------	-------		------------  	--------------------------------------------
2019/04/05 	0000.00	 	G.Cera 			Creation of the PRG

**********************************************************************************************************)

PROGRAM _csp_normal
VAR
END_VAR

csp();

_csp_case_normal();

_csp_transfer_normal();

_csp_main_normal();

_csp_customerInterfaces_normal();

END_PROGRAM

// ---- Application/CSP/Case/_Tasks/_csp_case_normal.TcPOU
(*********************************** G.D S.p.A. - Technical Department ***********************************
============= PROGRAM INFO ============
FOLDER:             TBD
MACHINES INVOLVED:  TBD 

============= DESCRIPTION =============
csp main interface program

============= REVISIONS ===============
Date		Version	 	Author      	Description             
----------	-------		------------  	--------------------------------------------
2019/09/27 	0000.00	 	M.Grasso		Creation of the PRG

**********************************************************************************************************)
PROGRAM _csp_case_normal
VAR
END_VAR

csp_case();

_csp_case_closing_normal();

_csp_case_discharge_normal();

_csp_case_feed_normal();

_csp_case_flapControl_normal();

_csp_case_glue_normal();

_csp_case_loader_normal();

_csp_case_openFlap_normal();

_csp_case_main_normal();

_csp_case_topRail_normal();

_csp_case_transport_normal();

END_PROGRAM

// ---- Application/CSP/Case/Closing/_Tasks/_csp_case_closing_normal.TcPOU
(*********************************** G.D S.p.A. - Technical Department ***********************************
============= PROGRAM INFO ============
FOLDER:             TBD
MACHINES INVOLVED:  TBD 

============= DESCRIPTION =============
csp main interface program

============= REVISIONS ===============
Date		Version	 	Author      	Description             
----------	-------		------------  	--------------------------------------------
2019/09/27 	0000.00	 	M.Grasso		Creation of the PRG

**********************************************************************************************************)
PROGRAM _csp_case_closing_normal
VAR
END_VAR

(* CASE *)
	(* CLOSING *)
		(* OS *)
		csp_case_closing_os();
	
		(* LS *)
		csp_case_closing_ls();

END_PROGRAM

// ---- Application/CSP/Case/Closing/OS/csp_case_closing_os.TcPOU
(*********************************** G.D S.p.A. - Technical Department ***********************************
============= PROGRAM INFO ============
FOLDER:             TBD
MACHINES INVOLVED:  TBD 

============= DESCRIPTION =============
csp machine declaration

============= REVISIONS ===============
Date		Version	 	Author      	Description             
----------	-------		------------  	--------------------------------------------
2019/04/05 	0000.00	 	M.Grasso		Creation of the PRG

**********************************************************************************************************)
(*$R process_ref := prc; $*)
PROGRAM csp_case_closing_os
VAR
		
	prc:											process;
	prc_path:										STRING;
	
	phase_upper:									BOOL;
	phase_lower:									BOOL;
	phase_horizontal:								BOOL;
	
	horizontal_first:								BOOL;
	horizontal_second:								BOOL;
	Closing_paddle_Cleanout_position_aem:			message;
	
END_VAR

VAR CONSTANT
	MOTOR_MAX_VELOCITY_DEGPS:							LREAL := 9600;
	MOTOR_MAX_ACCELLERATION_DEGPS2:						LREAL := 4800;
	MOTOR_MAX_DECELLERATION_DEGPS2:						LREAL := 4800;
	MOTOR_MAX_JERK_DEGPS3:								LREAL := 100000000; 
	MOTOR_MAX_FOLLOWING_ERROR_DEG:						LREAL := 2;
END_VAR

_read_var_input();

_object_manager();

IF NOT objects_running()
THEN
	RETURN;	
END_IF

_read_process_image();

_mode_manager();

_set_runtime_properties();

(********************************* BODY *********************************)

(* CLEARS PHASING SEQUENCE DUE TO AXES CAM ENGAGED *)
IF 	axis_is_cam_engaged(csp_case_closing_os_horizontal.axis)
	OR machine_is_stop_emergency_active(csp.mch)
THEN
	phase_horizontal := FALSE;
END_IF

IF 	axis_is_cam_engaged(csp_case_closing_os_upper.axis)
	OR machine_is_stop_emergency_active(csp.mch)
THEN
	phase_upper := FALSE;
END_IF

IF 	axis_is_cam_engaged(csp_case_closing_os_lower.axis)
	OR machine_is_stop_emergency_active(csp.mch)
THEN
	phase_lower := FALSE;
END_IF

IF (
	axis_is_cam_engaged(csp_case_closing_os_horizontal.axis)
	AND axis_is_cam_engaged(csp_case_closing_os_upper.axis)
	AND axis_is_cam_engaged(csp_case_closing_os_lower.axis)
	)
	OR machine_is_stop_emergency_active(csp.mch)
THEN
	horizontal_first := FALSE;
	horizontal_second := FALSE;
END_IF

(* HORIZONTAL NEEDS TO PHASE - CHECK IF UPPER AND LOWER MOVE FIRST OR HORIZONTAL FIRST *)
IF 	NOT axis_is_cam_engaged(csp_case_closing_os_horizontal.axis)
	AND NOT csp_case_closing_os_horizontal.phase_done
	AND (motorization_manager_is_starting(csp_main_motorization_manager.motm) OR jog_manager_is_jog_axis_active(JOG_LIST_CSP_CASE_VIRTUAL, csp_main_jogManager.jog_manager_virtual))
THEN	
	(* CALCULATED HORIZONTAL TO MOVE IN - MOVE UPPER AND LOWER FIRST *)
	IF csp_case_closing_os_horizontal.axis_calculated_cam_slave_position_deg >= axis_get_actual_modulo_position(csp_case_closing_os_horizontal.axis)
	THEN
		horizontal_second := TRUE;
	(* CALCULATED HORIZONTAL TO MOVE OUT - MOVE HORIZONTAL FIRST *)
	ELSE
		horizontal_first := TRUE;
	END_IF
END_IF
(* PHASE HORIZONTAL THEN UPPER AND LOWER *)
IF 	horizontal_first
	AND (motorization_manager_is_starting(csp_main_motorization_manager.motm) 
	OR jog_manager_is_jog_axis_active(JOG_LIST_CSP_CASE_VIRTUAL, csp_main_jogManager.jog_manager_virtual))
THEN
	phase_horizontal := TRUE;
	IF csp_case_closing_os_horizontal.phase_done
	THEN
		phase_upper := TRUE;
		phase_lower := TRUE;
	END_IF
END_IF
(* PHASE UPPER AND LOWER THEN HORIZONTAL *)
IF	horizontal_second
	AND (motorization_manager_is_starting(csp_main_motorization_manager.motm) 
	OR jog_manager_is_jog_axis_active(JOG_LIST_CSP_CASE_VIRTUAL, csp_main_jogManager.jog_manager_virtual))
THEN
	phase_upper := TRUE;
	phase_lower := TRUE;
	IF 	csp_case_closing_os_upper.phase_done
		AND csp_case_closing_os_lower.phase_done
	THEN
		phase_horizontal := TRUE;
	END_IF
END_IF

IF 	csp_case_closing.OS_Closing_Paddles_cleanout_position
	AND machine_is_ready(csp.mch)
THEN
	axis_enable(csp_case_closing_os_horizontal.axis);
	axis_enable(csp_case_closing_os_lower.axis);
	axis_enable(csp_case_closing_os_upper.axis);
END_IF
				
IF  csp_case_closing.OS_Closing_Paddles_cleanout_position
	AND axis_is_standstill(csp_case_closing_os_horizontal.axis)
	AND axis_is_standstill(csp_case_closing_os_lower.axis)
	AND axis_is_standstill(csp_case_closing_os_upper.axis)
THEN
	axis_move_absolute(
		position 		:= csp_case_closing_os_horizontal.accu_safe_pos,
		velocity 		:= 10,
		direction		:= AXIS_SHORTEST_WAY,
		acceleration 	:= MOTOR_MAX_ACCELLERATION_DEGPS2,
		deceleration 	:= MOTOR_MAX_DECELLERATION_DEGPS2,
		jerk 			:= MOTOR_MAX_JERK_DEGPS3, 
		buffer_mode 	:= AXIS_BUFFER_MODE_BUFFERED,
		CONVERSION_this := csp_case_closing_os_horizontal.axis); 
	axis_move_absolute(
		position 		:= csp_case_closing_os_lower.accu_safe_pos,
		velocity 		:= 5,
		direction		:= AXIS_SHORTEST_WAY,
		acceleration 	:= MOTOR_MAX_ACCELLERATION_DEGPS2,
		deceleration 	:= MOTOR_MAX_DECELLERATION_DEGPS2,
		jerk 			:= MOTOR_MAX_JERK_DEGPS3, 
		buffer_mode 	:= AXIS_BUFFER_MODE_BUFFERED,
		CONVERSION_this := csp_case_closing_os_lower.axis); 
	
	axis_move_absolute(
		position 		:= csp_case_closing_os_upper.accu_safe_pos,
		velocity 		:= 5,
		direction		:= AXIS_SHORTEST_WAY,
		acceleration 	:= MOTOR_MAX_ACCELLERATION_DEGPS2,
		deceleration 	:= MOTOR_MAX_DECELLERATION_DEGPS2,
		jerk 			:= MOTOR_MAX_JERK_DEGPS3, 
		buffer_mode 	:= AXIS_BUFFER_MODE_BUFFERED,
		CONVERSION_this := csp_case_closing_os_upper.axis); 			
END_IF

IF  csp_case_closing.OS_Closing_Paddles_cleanout_position
	AND csp_case_closing_os_upper.in_accu_safe_pos
	AND csp_case_closing_os_lower.in_accu_safe_pos
	AND csp_case_closing_os_horizontal.in_accu_safe_pos
THEN 
	process_message_set(1, 1, 1, Closing_paddle_Cleanout_position_aem);
END_IF


IF machine_is_stopped(csp.mch)
	OR machine_is_stop_emergency_active(csp.mch)
	AND NOT  csp_case_closing.OS_Closing_Paddles_cleanout_position
THEN
	process_message_reset(Closing_paddle_Cleanout_position_aem);		
END_IF



(************************************************************************)

_handle_messages();

_write_output();

ACTION _handle_messages:
;
END_ACTION

ACTION _handle_process_test:
;
END_ACTION

